20:	IF FSD.MODE = BYTE#0 THEN
		total_bytes := FSD.FILE_SIZE;
		X.NEW_FILE_SIZE := total_bytes + INT_TO_UDINT(idx);
		IF log_stop OR aw_aktiv THEN
			aw_aktiv := FALSE;
			FSD.MODE := BYTE#5; (* Datei schliessen *)
			(* ---------------- Debug-Message -----------------------*)
			(*IF _debug_enable THEN
				LOG_CL.NEW_MSG := 'FILE_XML2 - Close: [~2]';
				LOG_CL.PRINTF[2] := DT_TO_STRING(DTI);
				LOG_MSG();
			END_IF;*)
			(* -----------------------------------------------------------------*)
		END_IF;
		step_2 := 30;
	END_IF;

30:	IF FSD.MODE = BYTE#0 THEN (* Datei schliessen beendet *)
		IF log_stop THEN
			X.NEW_FILE_RTRIG := TRUE;
			log_stop := FALSE;
			SAVE_DATA.FN_REM := ''; (* remanenten Dateinamen löschen *)
		END_IF;
		step_2 := 00;
	END_IF;

END_CASE;

FS(FSD:=FSD,PT:=PT); (* FILE_SERVER *)

(* Fehlerauswertung *)
IF FSD.ERROR <> BYTE#0 THEN
	ERROR_C := BYTE_TO_DWORD(FSD.ERROR);
	ERROR_T := BYTE#1;
ELSIF X.UCB.BUF_DATA_LOST > UDINT#0 THEN
	ERROR_C := DWORD#2; (* Fehler: Bufferüberlauf - Datenmenge reduzieren *)
	ERROR_T := BYTE#6; 	(* Type: Buffer *)
ELSIF X.UCB.BUF_USED_MAX > USINT#90 THEN
	ERROR_C := DWORD#1; (* Warnung: Buffer auslastung > 90% *)
	ERROR_T := BYTE#6;	(* Type: Buffer *)
ELSE
	ERROR_C := DWORD#0;
	ERROR_T := BYTE#0;
END_IF;

trig_m_last := TRIG_M;

(* revision history
ks	25. july. 2011	rev 1.0
	original version

ks	16. apr. 2012	rev 1.1
	neuer überarbeiteter Code für automatisches File-open/close

ks	8. mar. 2016	rev 1.2
	nur einmal nach satellitenbausteinen scannen

ks	21. mar. 2016	rev 1.3
	prüfung auf freien bufferplatz hinzugefügt
	fehlermeldungen hinzugefügt

*)
          
END_FUNCTION_BLOCK

FUNCTION_BLOCK DLOG_STORE_MYSQL
  VAR_IN_OUT
    SQL_INFO : MYSQL_INFO;
    X : DLOG_DATA;
  END_VAR
  VAR_INPUT
    ENABLE : BOOL;
    TRIG_M : BOOL;
    TRIG_T : TIME;
    DTI : DT;
    URL : STRING(OSCAT_BASIC.STRING_LENGTH);
    DB_NAME : STRING(64);
    TB_NAME : STRING(64);
    AUTO_DELETE : UDINT;
    TIMEOUT : TIME;
    DNS_IP4 : DWORD;
  END_VAR
  VAR_OUTPUT
    ERROR_C : DWORD;
    ERROR_T : BYTE;
  END_VAR
  VAR
    UCB : UNI_CIRCULAR_BUFFER;
    MYSQL_CONTROL : MYSQL_CONTROL;
    trig_auto : BOOL;
    trig_tmp : BOOL;
    trig_m_last : BOOL;
    dti_last : DT := DATE_AND_TIME#2070-2-6-6:28:15;
    enable_last : BOOL;
    step : INT;
    idx : INT;
    n : USINT;
    snd_text : STRING(OSCAT_BASIC.STRING_LENGTH);
    snd_size : INT;
    sql_command : BYTE;
    next_step : INT;
    i1 : INT;
    i2 : INT;
    y : MYSQL_COM;
    del_dt : UDINT;
    del_start : BOOL;
    run : BOOL;
  END_VAR

            X.DTI := DTI; (* Datum / Zeit eintragen *)
X.CLOCK_TRIG := DTI <> dti_last;
dti_last := DTI;
trig_auto := FALSE;
IF X.CLOCK_TRIG THEN (* Impuls in jeder Sekunde *)
	del_start := DT_TO_UDINT(DTI) - del_dt > AUTO_DELETE AND AUTO_DELETE > UDINT#0;
	IF TRIG_T >= T#1000ms THEN (* automatischer Trigger *)
		trig_auto := DT_TO_UDINT(DTI) MOD (TIME_TO_UDINT(TRIG_T) / UDINT#1000) = UDINT#0;
	END_IF;
END_IF;
X.ADD_COM := 00;

CASE step OF

00:	IF ENABLE AND enable_last = FALSE THEN
		y.SQL_URL := URL;
		y.TIMEOUT := TIMEOUT;
		y.DNS_IP4 := DNS_IP4;
		y.SQL_CON := TRUE;

		X.UCB.D_MODE := 99; (* Buffer reset - Alles löschen *)
		UCB(DATA:=X.UCB);

		IF X.ID_MAX = USINT#0 THEN (* nur einmal nach Satellitenbausteinen scannen *)
			X.ADD_COM := 01; (* ADD INFO *)
			X.STORE_TYPE := BYTE#5; (* MySQL-Modus *)
		END_IF;

		step := 05;
	END_IF;

05:	X.ADD_COM := 02; (* ADD HEADER *)
	step := 10;

10:	IF SQL_INFO.SQL_CONNECTED THEN
		sql_command := BYTE#3; (* CREATE DATABASE IF NOT EXISTS `db_name` *)
		snd_text :=  CONCAT('CREATE DATABASE IF NOT EXISTS `' ,DB_NAME);
		snd_text :=  CONCAT(snd_text, '`');
		next_step := 20;
	END_IF;

20:	sql_command := BYTE#2; (* 0x02 COM_INIT_DB mysql_select_db *)
	snd_text := DB_NAME;
	next_step := 30;

30:	(* CREATE TABLE IF NOT EXISTS tb_name (Timestamp TIMESTAMP NULL DEFAULT CURRENT_TIMESTAMP, n1,n2) *)
	sql_command := BYTE#0;
	idx := 5;
	n := USINT#0;
	WHILE sql_command = BYTE#0 DO
		IF n = USINT#0 THEN
			snd_text := CONCAT('CREATE TABLE IF NOT EXISTS `', TB_NAME);
			snd_text := CONCAT(snd_text,'` (`ID` BIGINT NOT NULL AUTO_INCREMENT PRIMARY KEY ,');
			snd_text := CONCAT(snd_text,' store_timestamp TIMESTAMP NULL DEFAULT CURRENT_TIMESTAMP');
		ELSIF n <= X.ID_MAX THEN
			X.UCB.D_MODE := 12; (* Element lesen und löschen *)
			UCB(DATA:=X.UCB);
			snd_text := CONCAT(', `',X.UCB.D_STRING);
			CASE WORD_TO_INT(SHR(X.UCB.D_HEAD,8)) OF
			02:	snd_text := CONCAT(snd_text, '` FLOAT'); (* REAL *)
			06:	snd_text := CONCAT(snd_text, '` BOOL'); (* BOOL *)
			08:	snd_text := CONCAT(snd_text, '` INT'); (* DINT *)
			13:	snd_text := CONCAT(snd_text, '` DATETIME'); (* DT *)
			ELSE
				snd_text := CONCAT(snd_text, '` VARCHAR(80)'); (* STRING(80) *)
			END_CASE;
		ELSE
			snd_text := ')';
			sql_command := BYTE#3;
			snd_size := idx + LEN(snd_text);
			next_step := 40;
		END_IF;
		OSCAT_BASIC._STRING_TO_BUFFER(str:=snd_text,pos:=idx,pt:=ADR(y.S_BUF.BUFFER),size:=SIZEOF(y.S_BUF.BUFFER)); (* String in puffer kopieren *)
		idx := idx + LEN(snd_text);
		n := n + USINT#1;

		(*####################  DEBUG-MESSAGE  ###################################*)
		(*IF _debug_enable THEN
			LOG_CL.NEW_MSG := 'dlog_mysql: create >~1<';
			LOG_CL.PRINTF[1] := snd_text;
			LOG_MSG();
		END_IF;*)
		(*########################################################################*)
	END_WHILE;

40:	IF del_start THEN
		del_start := FALSE;
		sql_command := BYTE#3; (* DELETE FROM `tb_name` WHERE TIMESTAMPDIFF(SECOND, Timestamp, NOW()) > xxx *)
		snd_text := CONCAT('DELETE FROM `', TB_NAME);
		snd_text := CONCAT(snd_text, '` WHERE TIMESTAMPDIFF(SECOND, store_timestamp, NOW()) > ');
		snd_text := CONCAT(snd_text, UDINT_TO_STRING(AUTO_DELETE));
		next_step := 40;
		del_dt := DT_TO_UDINT(DTI);
		(*####################  DEBUG-MESSAGE  ###################################*)
		(*IF _debug_enable THEN
			LOG_CL.NEW_MSG := 'dlog_mysql: # delete time:~1 >~2<';
			LOG_CL.PRINTF[1] := UDINT_TO_STRING(AUTO_DELETE);
			LOG_CL.PRINTF[2] := snd_text;
			LOG_MSG();
		END_IF;*)
		(*########################################################################*)

         (* INSERT INTO `tb_name` VALUES (CURRENT_TIMESTAMP,  "n1","n2") *)
	ELSIF X.UCB.BUF_COUNT >= USINT_TO_INT(X.ID_MAX) AND step > 0 THEN (* Neue Datenreihe(n) vorhanden *)
		idx := 5;
		n := USINT#0;
		sql_command := BYTE#0;
		WHILE sql_command = BYTE#0 DO
			IF n = USINT#0 THEN
				snd_text := CONCAT('INSERT INTO `', TB_NAME);
				snd_text := CONCAT(snd_text,'` VALUES (NULL, CURRENT_TIMESTAMP');
			ELSIF n <= X.ID_MAX THEN
				X.UCB.D_MODE := 12; (* Element lesen und löschen *)
				UCB(DATA:=X.UCB);
				snd_text := CONCAT(', "',X.UCB.D_STRING);
				snd_text := CONCAT(snd_text, '"');
			ELSE
				snd_text := ')';
				sql_command := BYTE#3;
				snd_size := idx + LEN(snd_text);
				next_step := 40;
			END_IF;
			OSCAT_BASIC._STRING_TO_BUFFER(str:=snd_text,pos:=idx,pt:=ADR(y.S_BUF.BUFFER),size:=SIZEOF(y.S_BUF.BUFFER)); (* String in puffer kopieren *)
			idx := idx + LEN(snd_text);
			n := n + USINT#1;

			(*####################  DEBUG-MESSAGE  ###################################*)
			(*IF _debug_enable THEN
				LOG_CL.NEW_MSG := 'dlog_mysql: insert >~1<';
				LOG_CL.PRINTF[1] := snd_text;
				LOG_MSG();
			END_IF;*)
			(*########################################################################*)
		END_WHILE;
	END_IF;

	IF ENABLE THEN 	(* LOG-Trigger verarbeiten *)
		trig_tmp := (TRIG_M AND NOT trig_m_last) OR trig_auto OR X.ADD_DATA_REQ;

		IF trig_tmp THEN (* manueller, automatischer oder externer Trigger *)
			X.ADD_COM := 03; (* ADD DATA *)
			(* ---------------- Debug-Message -----------------------*)
			(*IF _debug_enable THEN
				LOG_CL.NEW_MSG := 'dlog_mysql: Trigger: DATE [~2]';
				LOG_CL.PRINTF[2] := DT_TO_STRING(DTI);
				LOG_MSG();
			END_IF;*)
			(* -----------------------------------------------------------------*)
		ELSE
			X.ADD_COM := 04;	(* ADD DATA REQ *)
		END_IF;
	ELSE
		y.SQL_CON := FALSE; (* MySQL Verbindung beenden *)
		step := 0;
	END_IF;
	X.ADD_DATA_REQ := FALSE;

(* ~~~~~~~~~~~~~~~~~~~~~~ *)

199:IF y.SQL_RCV_STATE = BYTE#1 THEN (* OK *)
		step := next_step;
	ELSIF y.SQL_RCV_STATE = BYTE#2 THEN  (* FEHLER *)
		step := 0;
	END_IF;

END_CASE;

(* ########################## *)
(* SQL-Kommando ausführen *)
IF sql_command > BYTE#0 THEN

	IF snd_size > 0 THEN
		y.S_BUF.SIZE := INT_TO_UINT(snd_size);
		snd_size := 0;
	ELSE
		OSCAT_BASIC._STRING_TO_BUFFER(str:=snd_text,pos:=5,pt:=ADR(y.S_BUF.BUFFER),size:=SIZEOF(y.S_BUF.BUFFER)); (* String in puffer kopieren *)
		y.S_BUF.SIZE := INT_TO_UINT(5 + LEN(snd_text));
		snd_text := '';
	END_IF;

	IF y.S_BUF.SIZE > SIZEOF(y.S_BUF.BUFFER) THEN (* buffer überlauf erkannt -> Abbruch *)
		y.S_BUF.SIZE := 0;
		sql_command := BYTE#0;
		y.SQL_CON := FALSE; (* MySQL Verbindung beenden *)
		step := 999; (* Dummy-Schritt *)
	ELSE

		i2 := UINT_TO_INT(y.S_BUF.SIZE) - 1; (* alle " zeichen mit ' ersetzen *)
		FOR i1 := 5 TO i2 DO
			IF y.S_BUF.BUFFER[i1] = BYTE#34 THEN
				y.S_BUF.BUFFER[i1] := BYTE#39;
			END_IF;
		END_FOR;
	
		y.S_BUF.BUFFER[4] := sql_command;
		y.SQL_PACKET_NO := BYTE#255;
		sql_command := BYTE#0;
		step := 199;
	END_IF;
END_IF;

(* ########################## *)

MYSQL_CONTROL(COM:= y, INFO:=SQL_INFO);

(* Fehlerauswertung *)
IF step = 999 THEN	(* Buffer überlauf *)
	ERROR_C := DWORD#3; (* Netzwerkbuffer überlauf *)
	ERROR_T := BYTE#6; 	(* Type: Buffer *)
ELSIF y.ERROR_T > BYTE#0 THEN	(* SQL Error *)
	ERROR_C := y.ERROR_C;
	ERROR_T := y.ERROR_T;
	step := 0;
ELSIF X.UCB.BUF_DATA_LOST > UDINT#0 THEN
	ERROR_C := DWORD#2; (* Fehler: Bufferüberlauf - Datenmenge reduzieren *)
	ERROR_T := BYTE#6; 	(* Type: Buffer *)
ELSIF X.UCB.BUF_USED_MAX > USINT#90 THEN
	ERROR_C := DWORD#1; (* Warnung: Buffer auslastung > 90% *)
	ERROR_T := BYTE#6;	(* Type: Buffer *)
ELSE
	ERROR_C := DWORD#0;
	ERROR_T := BYTE#0;
END_IF;



(* ########################## *)

trig_m_last := TRIG_M;
enable_last := ENABLE;
run := step > 0;

(* revision history
ks	20. apr. 2012	rev 1.0
	original version

ks	17. jan. 2014	rev 1.1
	DELTA Error 

ks	8. mar. 2016	rev 1.2
	nur einmal nach satellitenbausteinen scannen

ks	21. mar. 2016	rev 1.3
	prüfung auf bufferüberlauf und fehlermeldungen hinzugefügt

*)
          
END_FUNCTION_BLOCK

FUNCTION_BLOCK DLOG_STORE_RRD
  VAR_IN_OUT
    X : DLOG_DATA;
  END_VAR
  VAR_INPUT
    ENABLE : BOOL;
    TRIG_M : BOOL;
    TRIG_T : TIME;
    URL : STRING(OSCAT_BASIC.STRING_LENGTH);
    DTI : DT;
    SEP : BYTE;
    DNS_IP4 : DWORD;
    TIMEOUT : TIME;
  END_VAR
  VAR_OUTPUT
    ERROR_C : DWORD;
    ERROR_T : BYTE;
  END_VAR
  VAR
    UCB : UNI_CIRCULAR_BUFFER;
    IP_C : IP_C;  (* IP_Control Verwaltungsstruktur *)
    S_BUF : NETWORK_BUFFER;
    R_BUF : NETWORK_BUFFER;
    URL_DATA : url;
    DNS_CLIENT : DNS_CLIENT;
    HTTP_GET : HTTP_GET;
    IPC : IP_CONTROL;
    trig_auto : BOOL;
    trig_stored : BOOL;
    trig_tmp : BOOL;
    trig_m_last : BOOL;
    dti_last : DT := DATE_AND_TIME#2070-2-6-6:28:15;
    step_1 : INT;
    step_2 : INT;
    sep_char : STRING(1);
    url_query : STRING(OSCAT_BASIC.STRING_LENGTH);
    n : INT;
  END_VAR

            X.DTI := DTI; (* Datum / Zeit eintragen *)
X.CLOCK_TRIG := DTI <> dti_last;
dti_last := DTI;
trig_auto := FALSE;
IF X.CLOCK_TRIG THEN (* Impuls in jeder Sekunde *)
	IF TRIG_T >= T#1000ms THEN (* automatischer Trigger *)
		trig_auto := DT_TO_UDINT(DTI) MOD (TIME_TO_UDINT(TRIG_T) / UDINT#1000) = UDINT#0;
	END_IF;
END_IF;

CASE step_1 OF

00:	IF ENABLE THEN
		IF X.ID_MAX = USINT#0 THEN (* nur einmal nach Satellitenbausteinen scannen *)
			X.ADD_COM := 01; (* ADD INFO *)
			X.STORE_TYPE := BYTE#1; (* RRD-Modus *)
		END_IF;

		ERROR_T := BYTE#0;
		ERROR_C := DWORD#0;

		X.UCB.D_MODE := 99;
		UCB(DATA:=X.UCB); (* Buffer löschen *)

		URL_DATA:=STRING_TO_URL(STR:=URL,DEFAULT_PROTOCOL:='',DEFAULT_PATH:=''); (* URL zerlegen *)
		sep_char := OSCAT_BASIC.CHR_TO_STRING(SEP);
		url_query := URL_DATA.QUERY;
		step_1 := 30;

		(* ---------------- Debug-Message -----------------------*)
		(*IF _debug_enable THEN
			LOG_CL.NEW_MSG := 'FILE_RRD1 - Start: DATE [~2]';
			LOG_CL.PRINTF[2] := DT_TO_STRING(DTI);
			LOG_MSG();
		END_IF;*)
		(* -----------------------------------------------------------------*)

	END_IF;

30:	(* LOG-Trigger verarbeiten *)
	trig_tmp := (TRIG_M AND NOT trig_m_last) OR trig_auto OR X.ADD_DATA_REQ;

	IF ENABLE = FALSE THEN (* ENABLE = 0 -> Log Stop *)
		X.ADD_COM := 00;
		step_1 := 00;

		(* ---------------- Debug-Message -----------------------*)
		(*IF _debug_enable THEN
			LOG_CL.NEW_MSG := 'FILE_RRD1 - Stop: DATE [~2]';
			LOG_CL.PRINTF[2] := DT_TO_STRING(DTI);
			LOG_MSG();
		END_IF;*)
		(* -----------------------------------------------------------------*)

	ELSIF ENABLE THEN
		IF trig_tmp OR trig_stored THEN (* manueller, automatischer oder externer Trigger *)
			trig_stored := FALSE;
			X.ADD_COM := 03; (* ADD DATA *)
			(* ---------------- Debug-Message -----------------------*)
			(*IF _debug_enable THEN
				LOG_CL.NEW_MSG := 'FILE_RRD1 - Trig: DATE [~2]';
				LOG_CL.PRINTF[2] := DT_TO_STRING(DTI);
				LOG_MSG();
			END_IF;*)
			(* -----------------------------------------------------------------*)
		ELSE
			X.ADD_COM := 04;	(* ADD DATA REQ *)
		END_IF;
	END_IF;

END_CASE;
X.ADD_DATA_REQ := FALSE; (* externe Anforderung rücksetzen *)

(* ##################################### *)

CASE step_2 OF

00:	IF X.UCB.BUF_DATA_LOST > UDINT#0 THEN
		ERROR_C := DWORD#2; (* Fehler: Bufferüberlauf - Datenmenge reduzieren *)
		ERROR_T := BYTE#6; 	(* Type: Buffer *)
		step_2 := 100;
	ELSIF X.UCB.BUF_USED_MAX > USINT#90 THEN
		ERROR_C := DWORD#1; (* Warnung: Buffer auslastung > 90% *)
		ERROR_T := BYTE#6;	(* Type: Buffer *)
	END_IF;

	IF X.UCB.BUF_COUNT >= USINT_TO_INT(X.ID_MAX) THEN (* genug Einträge vorhanden *)
		URL_DATA.QUERY := url_query; (* original Query wiederherstellen *)
		n := 1;
		WHILE n <= USINT_TO_INT(X.ID_MAX) DO
			X.UCB.D_MODE := 12; (* Element lesen und löschen *)
			UCB(DATA:=X.UCB);
			IF n < USINT_TO_INT(X.ID_MAX) THEN (* Trennzeichen hinzufügen *)
				X.UCB.D_STRING := CONCAT(X.UCB.D_STRING,sep_char);
			END_IF;
			IF LEN(X.UCB.D_STRING) + LEN(URL_DATA.QUERY) <= OSCAT_BASIC.STRING_LENGTH THEN
				URL_DATA.QUERY := CONCAT(URL_DATA.QUERY,X.UCB.D_STRING); (* Query mit LOG-Daten ergänzen *)
				step_2 := 40;
			ELSE
				ERROR_T := BYTE#4; (* LOG-Daten können nicht in URL gepackt werden *)
				ERROR_C := DWORD#1;
				step_2 := 100;
			END_IF;
			n := n + 1;
		END_WHILE;;
	END_IF;

40:	IF DNS_CLIENT.DONE THEN
		step_2 := 60;
	ELSIF (DNS_CLIENT.ERROR > DWORD#0) THEN
		ERROR_C := DNS_CLIENT.ERROR; (* Fehlerbehandlung *)
		ERROR_T := BYTE#1;
		step_2 := 100;
	END_IF;

60:	IF HTTP_GET.DONE THEN
		n := UINT_TO_INT(HTTP_GET.BODY_START);
		IF R_BUF.BUFFER[n] <> BYTE#48 THEN (* ASCII '0' *)
			ERROR_C := DWORD#1;
			ERROR_T := BYTE#3;
		END_IF;
		step_2 := 100;

	ELSIF HTTP_GET.ERROR > DWORD#0 THEN (* Fehlerbehandlung *)
		ERROR_C := HTTP_GET.ERROR;
		ERROR_T := BYTE#2;
		step_2 := 100;
	END_IF;

100:	IF (NOT HTTP_GET.DONE) THEN (* UNLOCK HTTP DATA *)
		step_2 := SEL(ERROR_T = BYTE#0, 120,0);
	END_IF;

120:	IF NOT ENABLE THEN
		step_2 := 0;
	END_IF;

END_CASE;

HTTP_GET(IP_C:=IP_C,S_BUF:=S_BUF,R_BUF:=R_BUF,IP4:=DNS_CLIENT.IP4,GET:=step_2=60,MODE:=2,UNLOCK_BUF:=step_2=100,URL_DATA:=URL_DATA); (* HTTP_GET *)
DNS_CLIENT(IP_C:=IP_C, S_BUF:=S_BUF, R_BUF:=R_BUF, DOMAIN:=URL_DATA.DOMAIN, IP4_DNS:= DNS_IP4, ACTIVATE:=step_2=40); (* DNS-Client *)
IPC(IP:= 0, PORT:= 0 , TIME_OUT:= TIMEOUT, IP_C:= IP_C, S_BUF:= S_BUF, R_BUF:= R_BUF); (* IP_CONTROL *)

trig_m_last := TRIG_M;

(* revision history
ks	01. jan. 2011	rev 1.0
	original version

ks	13. may. 2011	rev 1.1
	ADD_DATA_REQ hinzugefügt

ks	26. july. 2011	rev 1.2
	code optimierung D_MODE 12 und bessere fehlerauswertung

ks	16. apr. 2012	rev 1.3
	neuer überarbeiteter Code

ks	21. mar. 2016	rev 1.4
	nur einmal nach satellitenbausteinen scannen und fehlermeldungen hinzugefügt

*)
          
END_FUNCTION_BLOCK

FUNCTION_BLOCK DLOG_STRING
  VAR_IN_OUT
    X : DLOG_DATA;
  END_VAR
  VAR_INPUT
    STR : STRING;
    COLUMN : STRING(40);
  END_VAR
  VAR
    UCB : UNI_CIRCULAR_BUFFER;
    id : WORD;
    str_last : STRING;
  END_VAR

            CASE x.ADD_COM OF

01:	(* ADD INFO *)
	X.ID_MAX := X.ID_MAX + USINT#1;
	id := WORD#16#0101; (* Quelltype STRING , Zieltype STRING *)
02:	(* ADD HEADER *)
	X.UCB.D_STRING := COLUMN;
	X.UCB.D_HEAD := id;
	X.UCB.D_MODE := 1;
	UCB(DATA:=X.UCB); (* Daten eintragen *)
03:	(* ADD DATA *)
	X.UCB.D_STRING := str_last;
	X.UCB.D_HEAD := id;
	X.UCB.D_MODE := 1;
	UCB(DATA:=X.UCB); (* Daten eintragen *)
END_CASE;
str_last := STR;

(* revision history
ks	01. jan. 2011	rev 1.0
	original version

ks	17. may. 2011	rev 1.1
	COLUMN STRING(40)

ks	25. july.   2011	rev 1.2
	neue head information

ks	19. apr.   2012	rev 1.3
	code neu überarbeitet
*)
          
END_FUNCTION_BLOCK

FUNCTION_BLOCK MYSQL_AUTH
  VAR_IN_OUT
    RUN : BOOL;
    PASSWORD : STRING(64);
    MESSAGE : ARRAY[0..19] OF BYTE;
    SCRAMBLE : ARRAY[0..19] OF BYTE;
  END_VAR
  VAR
    SHA1_STREAM : SHA1_STREAM;
    buf : ARRAY[0..63] OF BYTE;
    sha_mode : INT;
    step : INT;
    size : UDINT;
    pos : UDINT;
    i : INT;
    i2 : INT;
    scramble1 : ARRAY[0..19] OF BYTE;
    scramble2 : ARRAY[0..19] OF BYTE;
  END_VAR

            IF NOT RUN THEN RETURN; END_IF;
CASE step OF

0:	CASE sha_mode OF
	0:	sha_mode := 1; (* Initialisierung *)
		size := INT_TO_UDINT(LEN(PASSWORD));
		i2 := UDINT_TO_INT(size) - 1;
		FOR i := 0 TO 63 DO
			IF i <= i2 THEN
				buf[i] := OSCAT_BASIC.CODE(STR:=PASSWORD,POS:=i+1);
			ELSE
				buf[i] := BYTE#0;
			END_IF;
		END_FOR;

	3:	scramble1 := SCRAMBLE;
		sha_mode := 1; (* Initialisierung *)
		size := UDINT#20;
		FOR i := 0 TO 19 DO
			buf[i] := scramble1[i];
		END_FOR;
		step := 10;
	END_CASE;

10:	IF sha_mode = 3 THEN
		sha_mode := 1; (* Initialisierung *)
		scramble2 := SCRAMBLE;
		size := UDINT#40;
		FOR i := 0 TO 19 DO
			buf[i] := message[i];
			buf[i+20] := scramble2[i];
		END_FOR;
		step :=20;
	END_IF;

20:	IF sha_mode = 3 THEN
		sha_mode := 0; (* Stop *)
		FOR i:= 0 TO 19 DO
			SCRAMBLE[i] := SCRAMBLE[i] XOR scramble1[i];
		END_FOR;
		step :=0;
		RUN := FALSE;
	END_IF;
END_CASE;

SHA1_STREAM(SIZE:=size, MODE:=sha_mode, BUF:=buf, SHA1:=SCRAMBLE, POS=>pos);

(* revision history
ks	20. apr. 2012	rev 1.0
	original version

*)
          
END_FUNCTION_BLOCK

FUNCTION_BLOCK MYSQL_CONTROL
  VAR_IN_OUT
    COM : MYSQL_COM;
    INFO : MYSQL_INFO;
  END_VAR
  VAR
    IP_C : IP_C;
    URL_DATA : url;
    DNS_CLIENT : DNS_CLIENT;
    IPC : IP_CONTROL;
    step : INT;
    snd_step : INT;
    TON_WAIT : TON;
    last_step : INT;
    idx1 : INT;
    idx2 : INT;
    idx3 : INT;
    dw_tmp : DWORD;
    timeout1 : TIME;
    timeout2 : TIME;
    ip_c_red_disable : BOOL;
    auth_password : STRING(64);
    auth_run : BOOL;
    MYSQL_AUTH : MYSQL_AUTH;
    scramble1_buffer : ARRAY[0..19] OF BYTE;
    scramble2_buffer : ARRAY[0..19] OF BYTE;
    charset_number : BYTE := 16#8;
    max_packet_size : DWORD := 1024;
    client_flags : DWORD := 16#38601;
  END_VAR

            CASE step OF

00:	IF COM.SQL_CON THEN
		timeout1 := MAX(T#10s,COM.TIMEOUT);
		timeout2 := timeout1 + T#1s;
		INFO.SQL_ERROR := '';
		COM.ERROR_C := DWORD#0;
		COM.ERROR_T := BYTE#0;
		URL_DATA := STRING_TO_URL(STR:=COM.SQL_URL,DEFAULT_PROTOCOL:='',DEFAULT_PATH:='/');
		step := 10;
	END_IF;

10:	IF DNS_CLIENT.DONE THEN
		step := 20;
	ELSIF DNS_CLIENT.ERROR <> DWORD#0 THEN
		COM.ERROR_C := DNS_CLIENT.ERROR;
		COM.ERROR_T := BYTE#1;
		step := 980;
	END_IF;

20:	(* MySQL Steuerkanal einrichten *)
	IF URL_DATA.PORT = WORD#0 THEN
		URL_DATA.PORT := WORD#3306; (* Standard Port *)
	END_IF;
	IP_C.C_PORT := URL_DATA.PORT; (* Portnummer eintragen *)
  	IP_C.C_IP := DNS_CLIENT.IP4; (* IP eintragen *)
  	IP_C.C_MODE := BYTE#0; (* Mode: TCP+ACTIV+PORT *)
  	IP_C.TIME_RESET := TRUE; (* Zeitueberwachung rücksetzen *)
  	IP_C.C_ENABLE := TRUE; (* Verbindungsaufbau freigeben *)
  	IP_C.R_OBSERVE := TRUE; (* Empfangsueberwachung *)
	COM.R_BUF.SIZE := UINT#0;
	COM.SQL_RCV_STATE := BYTE#0;
	step := 30;

30:	IF COM.SQL_RCV_STATE = BYTE#1 THEN
		INFO.SERVER_PROTOCOL_VERSION := COM.R_BUF.BUFFER[4];

		(* ende markierung von string server_version suchen *)
		idx2 := UINT_TO_INT(COM.R_BUF.SIZE) - 1;
		FOR idx1 := 5 TO idx2 DO
			IF COM.R_BUF.BUFFER[idx1] = BYTE#0 THEN EXIT; END_IF;
		END_FOR;
		idx1 := idx1 + 5; (* terminierung und thread-id überspringen *)

		FOR idx2:=0 TO 7 DO	(* Byte 0-7 *)
			scramble1_buffer[idx2] := COM.R_BUF.BUFFER[idx1];
			idx1 := idx1 + 1;
		END_FOR;
		idx1 := idx1 + 1;
		idx2 := idx1 + 1;
		INFO.SERVER_CAPABILITIES := OSCAT_BASIC.WORD_OF_BYTE(COM.R_BUF.BUFFER[idx2], COM.R_BUF.BUFFER[idx1]);
		idx1 := idx1 + 2;
		INFO.SERVER_LANGUAGE := COM.R_BUF.BUFFER[idx1];
		idx1 := idx1 + 1;
		idx2 := idx1 + 1;
		INFO.SERVER_STATUS := OSCAT_BASIC.WORD_OF_BYTE(COM.R_BUF.BUFFER[idx2], COM.R_BUF.BUFFER[idx1]);
		idx1 := idx1 + 15;

		FOR idx2:=8 TO 19 DO	(* Byte 8-19 *)
			scramble1_buffer[idx2] := COM.R_BUF.BUFFER[idx1];
			idx1 := idx1 + 1;
		END_FOR;

		IF INFO.SERVER_PROTOCOL_VERSION < BYTE#10 THEN  (* Error: protocol version zu niedrig *)
			COM.ERROR_T := BYTE#2;
			COM.ERROR_C := DWORD#1;
			step := 980;
		ELSIF URL_DATA.PASSWORD = '' THEN
			step := 50;
		ELSE
			auth_password := URL_DATA.PASSWORD;
			auth_run := TRUE;
			step := 40;
		END_IF;
	END_IF;

40:	MYSQL_AUTH(RUN:= auth_run,PASSWORD:= auth_password ,MESSAGE:= scramble1_buffer,SCRAMBLE:= scramble2_buffer);
	IF NOT auth_run THEN
		step := 50;
	END_IF;

50: (* Client Authentication Packet *)
	(* Byte 0-3 werden später eingetragen *)
	COM.S_BUF.BUFFER[04] := OSCAT_BASIC.BYTE_OF_DWORD(client_flags, BYTE#0); (* client_flags *)
	COM.S_BUF.BUFFER[05] := OSCAT_BASIC.BYTE_OF_DWORD(client_flags, BYTE#1);
	COM.S_BUF.BUFFER[06] := OSCAT_BASIC.BYTE_OF_DWORD(client_flags, BYTE#2);
	COM.S_BUF.BUFFER[07] := OSCAT_BASIC.BYTE_OF_DWORD(client_flags, BYTE#3);
	COM.S_BUF.BUFFER[08] := OSCAT_BASIC.BYTE_OF_DWORD(max_packet_size, BYTE#0); (* max_packet_size *)
	COM.S_BUF.BUFFER[09] := OSCAT_BASIC.BYTE_OF_DWORD(max_packet_size, BYTE#1);
	COM.S_BUF.BUFFER[10] := OSCAT_BASIC.BYTE_OF_DWORD(max_packet_size, BYTE#2);
	COM.S_BUF.BUFFER[11] := OSCAT_BASIC.BYTE_OF_DWORD(max_packet_size, BYTE#3);
	COM.S_BUF.BUFFER[12] := charset_number; (* charset_number *)
	FOR idx1 := 13 TO 35 DO (* 23 bytes filler always 0x00.. *)
		COM.S_BUF.BUFFER[idx1] := BYTE#0;
	END_FOR;
	idx3 := LEN(URL_DATA.USER);
	FOR idx2 :=1 TO idx3 DO
		COM.S_BUF.BUFFER[idx1] := OSCAT_BASIC.CODE(URL_DATA.USER, idx2);
		idx1 := idx1 + 1;
	END_FOR;
	COM.S_BUF.BUFFER[idx1] := BYTE#0; (* String terminierung eintragen *)
	idx1 := idx1 + 1;
	IF LEN(URL_DATA.PASSWORD) = 0 THEN
		COM.S_BUF.BUFFER[idx1] := BYTE#0; (* scramble_buff length *)
	ELSE
		COM.S_BUF.BUFFER[idx1] := BYTE#20; (* scramble_buff length *)
		FOR idx2 :=0 TO 19 DO
			idx1 := idx1 + 1;
			COM.S_BUF.BUFFER[idx1] := scramble2_buffer[idx2];
		END_FOR;
	END_IF;
	COM.S_BUF.SIZE  := INT_TO_UINT(idx1 + 1); (* Sendelänge eintragen *)

	step := 60;

60:	IF COM.SQL_RCV_STATE = BYTE#1 THEN
		INFO.SQL_CONNECTED := TRUE;
		step := 300;
	END_IF;

(* ================================================== *)

300:	step := SEL(COM.SQL_CON,700,310); (* Schritt-Selektion *)

310:	step := 300; (* dummy step *)

(* ================================================== *)

700: (* COM_QUIT *)
	COM.S_BUF.BUFFER[04] := BYTE#1; (* 0x01 COM_QUIT mysql_close *)
	COM.S_BUF.SIZE := UINT#5; (* Sendelänge eintragen *)
	COM.SQL_PACKET_NO := BYTE#255;
	ip_c_red_disable := TRUE;
	step := 710;

710:	IF IP_C.C_STATE = BYTE#0 THEN (* Verbindung durch SQL-Server beendet ? *)
		step := 980;
	END_IF;

(* ================================================== *)

980:IP_C.C_ENABLE := FALSE; (* MYSQL Steuerkanal schliessen *)
	ip_c_red_disable := FALSE;
	INFO.SQL_CONNECTED := FALSE;
	COM.SQL_CON := FALSE;
	COM.S_BUF.SIZE := UINT#0;
	COM.R_BUF.SIZE := UINT#0;
	snd_step := 0;
	step := 990;
	(*####################  DEBUG-MESSAGE  ###################################*)
	(*IF _debug_enable THEN
		LOG_CL.NEW_MSG := 'QUIT: ERROR CODE >~1< TYPE >~2<';
		LOG_CL.PRINTF[1] := DWORD_TO_STRH(COM.ERROR_C);
		LOG_CL.PRINTF[2] := BYTE_TO_STRING(COM.ERROR_T);
		LOG_MSG();
	END_IF;*)
	(*########################################################################*)

990:IF IP_C.C_STATE = BYTE#0 THEN
		step := 0;
	END_IF;

END_CASE;

(* ++++++++++++++++++++++++++++++++++++++++++++++++++++++++++ *)

IF step >= 30 THEN
	IF COM.R_BUF.SIZE >= UINT#3 AND COM.SQL_RCV_STATE = BYTE#0 THEN (* Daten wurden empfangen ? *)
		IF DWORD_TO_UINT(OSCAT_BASIC.DWORD_OF_BYTE(BYTE#0, COM.R_BUF.BUFFER[2], COM.R_BUF.BUFFER[1], COM.R_BUF.BUFFER[0])) + UINT#4 = COM.R_BUF.SIZE THEN
			COM.SQL_PACKET_NO := COM.R_BUF.BUFFER[3];
			IF COM.R_BUF.BUFFER[4] = BYTE#16#FF THEN
				idx2 := 13; (* Error String - Erstes Zeichen *)
				idx3 := UINT_TO_INT(COM.R_BUF.SIZE) - 1; (* Error String - Letztes Zeichen *)
				FOR idx1 := idx2 TO idx3 DO (* alle ' durch ´ ersetzen *)
					IF COM.R_BUF.BUFFER[idx1] = BYTE#39 THEN
						COM.R_BUF.BUFFER[idx1] := BYTE#96;
					END_IF;
				END_FOR;
				INFO.SQL_ERROR := OSCAT_BASIC.BUFFER_TO_STRING(PT:=ADR(COM.R_BUF.BUFFER),SIZE:=COM.R_BUF.SIZE,START:=INT_TO_UINT(idx2),STOP:=INT_TO_UINT(idx3));
				COM.ERROR_T := BYTE#3;
				COM.ERROR_C := OSCAT_BASIC.DWORD_OF_BYTE(BYTE#0,BYTE#0,COM.R_BUF.BUFFER[6], COM.R_BUF.BUFFER[5]);
				COM.SQL_RCV_STATE := BYTE#2;
				COM.R_BUF.SIZE := UINT#0; (* Empfangsbuffer nach Fehler rücksetzen *)
				step := 980;
			ELSE
				COM.SQL_RCV_STATE := BYTE#1;
				IP_C.R_OBSERVE := FALSE;

				(*####################  DEBUG-MESSAGE  ###################################*)
				(*IF _debug_enable THEN
					LOG_CL.NEW_MSG := 'RCV: size >~1<';
					LOG_CL.PRINTF[1] := UINT_TO_STRING(COM.R_BUF.SIZE);
					LOG_MSG();
				END_IF;*)
				(*########################################################################*)
			END_IF;
		END_IF;
	END_IF;
END_IF;

(* automatisches Datensenden *)

CASE snd_step OF

00:	IF step >= 20 AND COM.S_BUF.SIZE > UINT#0 THEN
		dw_tmp := UINT_TO_DWORD(COM.S_BUF.SIZE - UINT#4); (* packet_length *)
		COM.S_BUF.BUFFER[0] := OSCAT_BASIC.BYTE_OF_DWORD(dw_tmp, BYTE#0);
		COM.S_BUF.BUFFER[1] := OSCAT_BASIC.BYTE_OF_DWORD(dw_tmp, BYTE#1);
		COM.S_BUF.BUFFER[2] := 0;
		COM.SQL_PACKET_NO := COM.SQL_PACKET_NO + 1;
		COM.S_BUF.BUFFER[3] := COM.SQL_PACKET_NO;

		IP_C.R_OBSERVE := TRUE;
		COM.R_BUF.SIZE := UINT#0; (* Empfangsbuffer rücksetzen *)
		COM.SQL_RCV_STATE := BYTE#0;

	        (*####################  DEBUG-MESSAGE  ###################################*)
	        (*IF _debug_enable THEN
	          LOG_CL.NEW_MSG := 'SND: size >~1<';
	          LOG_CL.PRINTF[1] := UINT_TO_STRING(COM.S_BUF.SIZE);
	          LOG_MSG();
	        END_IF;*)
	        (*########################################################################*)

		snd_step := 10;
	END_IF;

10:	IF COM.S_BUF.SIZE = UINT#0 THEN (* warten bis alle daten gesendet sind *)
		snd_step := 0;
	END_IF;

END_CASE;

(* Globale Fehlerbehandlung für Haupt-Routine *)
IF COM.ERROR_T = BYTE#0 AND step > 20 THEN (* noch kein Fehler gespeichert und Hauptroutine aktiv *)
	IF IP_C.ERROR > DWORD#0 AND IP_C.C_ENABLE AND NOT IP_C.TIME_RESET THEN  (* IP Control *)
		IF ip_c_red_disable = FALSE OR IP_C.ERROR <> DWORD#16#FD000000 THEN
			COM.ERROR_C := IP_C.ERROR;
			COM.ERROR_T := BYTE#2;
			step := 980;
		END_IF;
	END_IF;
END_IF;

IF TON_WAIT.Q THEN (* Ablaufstörung - Schrittkette *)
	COM.ERROR_C := INT_TO_DWORD(step); (* aktuellen Schritt eintragen *)
	COM.ERROR_T := BYTE#5;
	step := 980;
END_IF;

(* ######################################################## *)

DNS_CLIENT(IP_C:=IP_C, S_BUF:=COM.S_BUF, R_BUF:=COM.R_BUF, DOMAIN:=URL_DATA.DOMAIN, IP4_DNS:= COM.DNS_IP4, ACTIVATE:=step=10); (* DNS-Client *)
IPC(IP:= DWORD#0, PORT:= WORD#0 , TIME_OUT:= timeout1, IP_C:= IP_C, S_BUF:= COM.S_BUF, R_BUF:= COM.R_BUF); (* MYSQL Steuerkanal *)

TON_WAIT(IN:=step = last_step AND step > 0,PT:=timeout2);
last_step := step;

(* revision history
ks	20. apr. 2012	rev 1.0
	original version
ks	14. oct. 2013	rev 1.1
	DNS_CLIENT Fehler durch zugriffskonflikt zwischen dns_client und mySQL auf S_BUF

*)
          
END_FUNCTION_BLOCK

PROGRAM BASE64_DEMO
  VAR
    text1 : STRING(144) := '<4036.1076324381@guildenstern.zeitform.de>';
    text2 : STRING(192);
    text3 : STRING(144);
    BASE64_DECODE_STR : BASE64_DECODE_STR;
    BASE64_ENCODE_STR : BASE64_ENCODE_STR;
    start : BOOL := TRUE;
    done1 : BOOL;
    done2 : BOOL;
  END_VAR

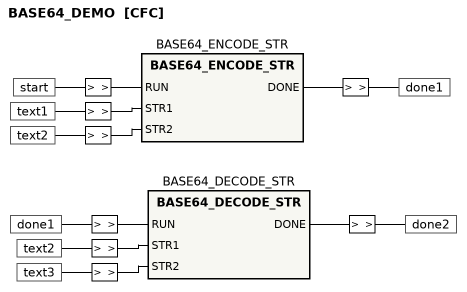
(* CFC diagram, written out as Structured Text *)
BASE64_ENCODE_STR(RUN := start, STR1 := text1, STR2 := text2);
done1 := BASE64_ENCODE_STR.DONE;
BASE64_DECODE_STR(RUN := done1, STR1 := text2, STR2 := text3);
done2 := BASE64_DECODE_STR.DONE;
END_PROGRAM

PROGRAM CSV_PARSER_BUF_DEMO
  VAR CONSTANT
    line_cnt : INT := 2;
    col_cnt : INT := 4;
  END_VAR
  VAR
    CPB : CSV_PARSER_BUF;
    FS : FILE_SERVER;
    FSD : FILE_SERVER_DATA;
    PT : NETWORK_BUFFER;
    sep : BYTE;
    value : STRING(OSCAT_BASIC.STRING_LENGTH);
    step : INT;
    result : BYTE;
    offset : UDINT;
    run : BYTE;
    done : BOOL;
    value_real : REAL;
    cnt : INT;
    line : INT;
    idx : INT;
    data : ARRAY[1..line_cnt, 1..col_cnt] OF REAL;
  END_VAR

            (* Demo-Programm: CSV-Datei mittels Enumeration auswerten
die groesse des arrays kann mittels konstanten line_cnt und col_cnt angepasst werden

 ----- den nachfolgenden Textblock als datei "csv.txt" auf der sps ablegen ---
10.45,20,30,40.8
115,3450.2123,456,123.1
---------------------------------------------------------------------------------*)

CASE step OF

00:	IF NOT done THEN
	 	(* File_Daten einrichten  *)
		FSD.FILENAME := 'csv.txt'; (* Dateiname *)
		FSD.MODE := 1; (* vorhandene Datei zum lesen öffnen *)
		FSD.OFFSET := 0; (* Start bei Dateianfang *)
		PT.SIZE := 65535; (* maximale länge einlesen *)
		step := 10;
	END_IF;

10:	IF FSD.MODE = 0 THEN (* Datei geöffnet ? *)
		OFFSET := 0; (* Start Offset vorgeben *)
		sep :=44; (* Trennzeichen , *)
		run := 1; (* Element suchen *)
		cnt := 0;
		step := 20;
	END_IF;

20:	IF run = 0 THEN
		(* ---------------------- Debug-Message ----------------------------*)
		(*IF _debug_enable THEN
			LOG_CL.NEW_MSG := 'CPFD: /value >~2< /offset ~3 /Run ~4 /Result ~5';
			LOG_CL.PRINTF[2] := value;
			LOG_CL.PRINTF[3] := UDINT_TO_STRING(OFFSET);
			LOG_CL.PRINTF[4] := BYTE_TO_STRING(run);
			LOG_CL.PRINTF[5] := BYTE_TO_STRING(result);
			LOG_MSG();
		END_IF;*)
		(* -----------------------------------------------------------------*)

		run := 1; (*  nächstes Element suchen  *)

		IF result = 1 OR result = 2 THEN
			(* automatische konvertierung in real ausführen *)
			IF LEN(value) <= 20 THEN
				value_real := OSCAT_BASIC.FLOAT_TO_REAL(FLT:=value);
			ELSE
				value_real := 0.0;
			END_IF;

			cnt := cnt + 1;
			IF cnt <= line_cnt * col_cnt THEN
				line := (cnt / col_cnt) + 1;
				idx := (cnt MOD col_cnt);
				data[line,idx] := value_real; (* Daten in Array eintragen *)
			END_IF;

		ELSIF result = 10 THEN (* nichts mehr gefunden *)
			run := 0; (* keine weitere INI Auswertung erwünscht *)
			FSD.MODE := 5; (* Datei schliessen *)
			step := 30;
		END_IF;
	END_IF;

30:	IF FSD.MODE = 0 THEN (* Datei geschlossen ? *)
		step := 0;
		done := TRUE;
	END_IF;

END_CASE;

CPB(SEP:=sep,RUN:=run,OFFSET:=OFFSET,VALUE:=value,PT:=PT,RESULT=>result); (* CSV PARAMETER BUF *)
FS(FSD:=FSD,PT:=PT); (* FILE_SERVER *)
          
END_PROGRAM

PROGRAM CSV_PARSER_FILE_DEMO
  VAR CONSTANT
    line_cnt : INT := 2;
    col_cnt : INT := 4;
  END_VAR
  VAR
    CPF : CSV_PARSER_FILE;
    FS : FILE_SERVER;
    FSD : FILE_SERVER_DATA;
    PT : NETWORK_BUFFER;
    filename : STRING;
    value : STRING(OSCAT_BASIC.STRING_LENGTH);
    sep : BYTE;
    step : INT;
    result : BYTE;
    offset : UDINT;
    run : BYTE;
    done : BOOL;
    value_real : REAL;
    cnt : INT;
    line : INT;
    idx : INT;
    data : ARRAY[1..line_cnt, 1..col_cnt] OF REAL;
  END_VAR

            (* Demo-Programm: CSV-Datei mittels Enumeration auswerten

die groesse des arrays kann mittels konstanten line_cnt und col_cnt angepasst werden

 ----- den nachfolgenden Textblock als datei "csv.txt" auf der sps ablegen ---
10.45,20,30,40.8
115,3450.2123,456,123.1
---------------------------------------------------------------------------------*)

CASE step OF

00:	IF NOT done THEN
		filename := 'csv.txt'; (* File_Daten einrichten *)
		OFFSET := 0; (* Start Offset vorgeben *)
		sep :=44; (* Trennzeichen , *)
		run := 1; (* Element suchen *)
		cnt := 0;
		step := 20;
	END_IF;

20:	IF run = 0 THEN (* kein Befehl mehr aktiv ? *)
		(* ---------------------- Debug-Message ----------------------------*)
		(*IF _debug_enable THEN
			LOG_CL.NEW_MSG := 'CPFD: /value >~2< /offset ~3 /Run ~4 /Result ~5';
			LOG_CL.PRINTF[2] := value;
			LOG_CL.PRINTF[3] := UDINT_TO_STRING(OFFSET);
			LOG_CL.PRINTF[4] := BYTE_TO_STRING(run);
			LOG_CL.PRINTF[5] := BYTE_TO_STRING(result);
			LOG_MSG();
		END_IF;*)
		(* -----------------------------------------------------------------*)

		run := 1; (*  nächstes Element suchen  *)

		IF result = 1 OR result = 2 THEN
			(* automatische konvertierung in real ausführen *)
			IF LEN(value) <= 20 THEN
				value_real := OSCAT_BASIC.FLOAT_TO_REAL(FLT:=value);
			ELSE
				value_real := 0.0;
			END_IF;

			cnt := cnt + 1;
			IF cnt <= line_cnt * col_cnt THEN
				line := (cnt / col_cnt) + 1;
				idx := (cnt MOD col_cnt);
				data[line,idx] := value_real; (* Daten in Array eintragen *)
			END_IF;

		ELSIF result = 10 THEN (* nichts mehr gefunden *)
			run := 0; (* keine weitere INI Auswertung erwünscht *)
			FSD.MODE := 5; (* Datei schliessen *)
			step := 30;
		END_IF;
	END_IF;

30:	IF FSD.MODE = 0 THEN (* Befehl Datei schliessen beendet *)
		step := 0;
		done := TRUE;
	END_IF;

END_CASE;

CPF(SEP:=sep,FILENAME:=FILENAME,FSD:=FSD,RUN:=run,OFFSET:=OFFSET,VALUE:=value,PT:=PT,RESULT=>result); (* CSV PARAMETER FILE *)
FS(FSD:=FSD,PT:=PT); (* FILE_SERVER *)
          
END_PROGRAM

PROGRAM DLOG_FILE_CSV_DEMO
  VAR
    cur_dt : DT;
    enable : BOOL := TRUE;
    trig_t : TIME := TIME#5s0ms;
    trig_m : BOOL;
    error_c : DWORD;
    error_t : BYTE;
    auto_close : TIME := TIME#10s0ms;
    x1 : DLOG_DT;
    x2 : DLOG_REAL;
    x3 : DLOG_DINT;
    x4 : DLOG_BOOL;
    x5 : DLOG_STRING;
    x : DLOG_DATA;
    RTC_2 : oscat_basic.RTC_2;
    DLOG_STORE_FILE_CSV : DLOG_STORE_FILE_CSV;
    GEN_SIN_1 : oscat_basic.GEN_SIN;
    COUNT_DR : oscat_basic.COUNT_DR;
  END_VAR
  VAR RETAIN
    save_data : DLOG_SAVE;
  END_VAR

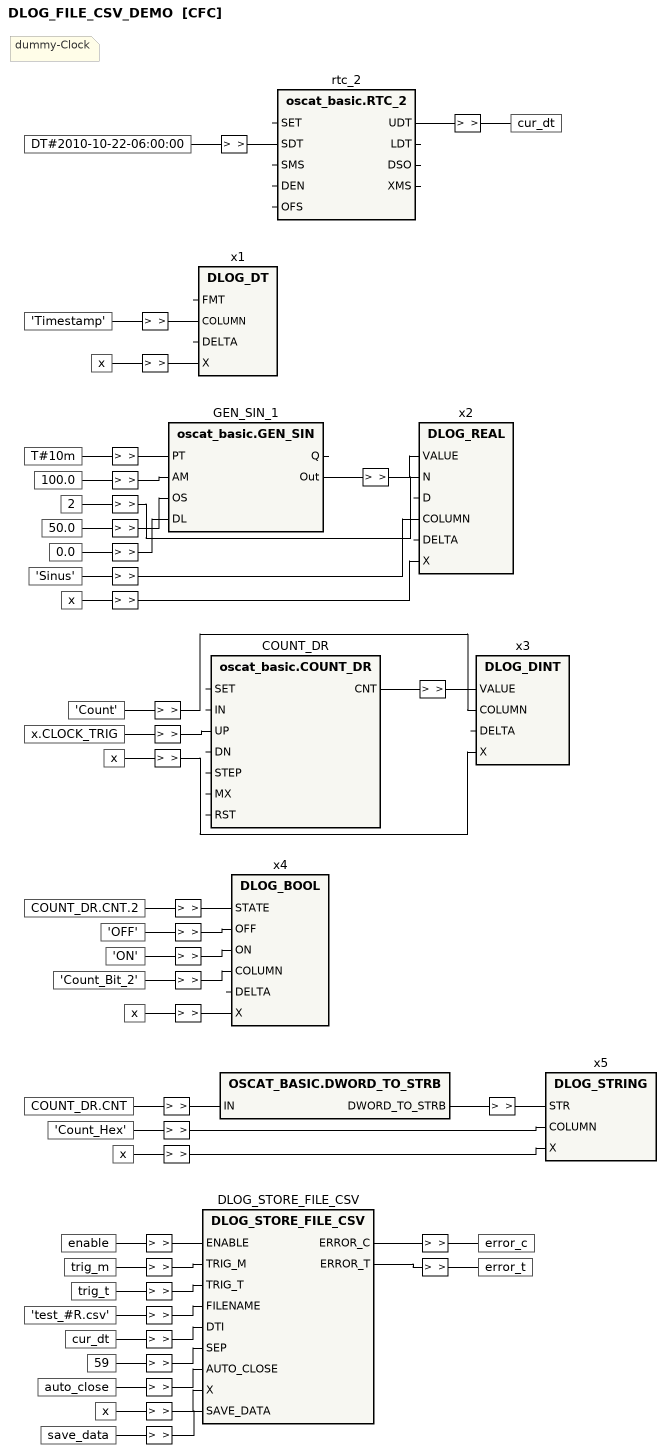
(* CFC diagram, written out as Structured Text *)
(* dummy-Clock *)
rtc_2(SDT := DT#2010-10-22-06:00:00);
cur_dt := rtc_2.UDT;
x1(COLUMN := 'Timestamp', X := x);
GEN_SIN_1(PT := T#10m, AM := 100.0, OS := 50.0, DL := 0.0);
x2(VALUE := GEN_SIN_1.Out, N := 2, COLUMN := 'Sinus', X := x);
COUNT_DR(UP := x.CLOCK_TRIG);
x3(VALUE := COUNT_DR.CNT, COLUMN := 'Count', X := x);
x4(STATE := COUNT_DR.CNT.2, OFF := 'OFF', ON := 'ON', COLUMN := 'Count_Bit_2', X := x);
x5(STR := OSCAT_BASIC.DWORD_TO_STRB(COUNT_DR.CNT), COLUMN := 'Count_Hex', X := x);
DLOG_STORE_FILE_CSV(ENABLE := enable, TRIG_M := trig_m, TRIG_T := trig_t, FILENAME := 'test_#R.csv', DTI := cur_dt, SEP := 59, AUTO_CLOSE := auto_close, X := x, SAVE_DATA := save_data);
error_c := DLOG_STORE_FILE_CSV.ERROR_C;
error_t := DLOG_STORE_FILE_CSV.ERROR_T;
END_PROGRAM

PROGRAM DLOG_FILE_CSV_FTP_DEMO
  VAR
    cur_dt : DT;
    enable : BOOL := TRUE;
    trig_t : TIME := TIME#5s0ms;
    trig_m : BOOL;
    error_c : DWORD;
    error_t : BYTE;
    auto_close : TIME := TIME#10s0ms;
    x1 : DLOG_DT;
    x2 : DLOG_REAL;
    x3 : DLOG_DINT;
    x4 : DLOG_BOOL;
    x5 : DLOG_STRING;
    x : DLOG_DATA;
    RTC_2 : oscat_basic.RTC_2;
    DLOG_STORE_FILE_CSV : DLOG_STORE_FILE_CSV;
    GEN_SIN_1 : oscat_basic.GEN_SIN;
    COUNT_DR : oscat_basic.COUNT_DR;
    DLOG_FILE_TO_FTP : DLOG_FILE_TO_FTP;
    ftp_done : BOOL;
    ftp_busy : BOOL;
    ftp_error_c : DWORD;
    ftp_error_t : BYTE;
    ftp_url : STRING := 'ftp://581920:123456@oscat.atwebpages.com:2000/subordner/';
    ftp_activ : BOOL := FALSE;
    ftp_delete : BOOL := TRUE;
    ftp_retry : INT := 0;
    ftp_retry_time : TIME := TIME#1m0s0ms;
    ftp_timeout : TIME := TIME#30s0ms;
  END_VAR
  VAR RETAIN
    save_data : DLOG_SAVE;
  END_VAR

(* CFC diagram, written out as Structured Text *)
(* dummy-Clock *)
rtc_2(SDT := DT#2010-10-22-06:00:00);
cur_dt := rtc_2.UDT;
x1(COLUMN := 'Timestamp', X := x);
GEN_SIN_1(PT := T#10m, AM := 100.0, OS := 50.0, DL := 0.0);
x2(VALUE := GEN_SIN_1.Out, N := 2, COLUMN := 'Sinus', X := x);
COUNT_DR(UP := x.CLOCK_TRIG);
x3(VALUE := COUNT_DR.CNT, COLUMN := 'Count', X := x);
x4(STATE := COUNT_DR.CNT.2, OFF := 'OFF', ON := 'ON', COLUMN := 'Count_Bit_2', X := x);
x5(STR := OSCAT_BASIC.DWORD_TO_STRB(COUNT_DR.CNT), COLUMN := 'Count_Hex', X := x);
DLOG_STORE_FILE_CSV(ENABLE := enable, TRIG_M := trig_m, TRIG_T := trig_t, FILENAME := 'test_#R.csv', DTI := cur_dt, SEP := 59, AUTO_CLOSE := auto_close, X := x, SAVE_DATA := save_data);
error_c := DLOG_STORE_FILE_CSV.ERROR_C;
error_t := DLOG_STORE_FILE_CSV.ERROR_T;
DLOG_FILE_TO_FTP(FTP_URL := ftp_url, FTP_ACTIV := ftp_activ, FILE_DELETE := ftp_delete, TIMEOUT := ftp_timeout, RETRY := ftp_retry, RETRY_TIME := ftp_retry_time, DNS_IP4 := oscat_basic.DWORD_OF_BYTE(8, 8, 8, 8), PLC_IP4 := oscat_basic.DWORD_OF_BYTE(192, 168, 178, 025), X := x);
ftp_done := DLOG_FILE_TO_FTP.DONE;
ftp_busy := DLOG_FILE_TO_FTP.BUSY;
ftp_error_c := DLOG_FILE_TO_FTP.ERROR_C;
ftp_error_t := DLOG_FILE_TO_FTP.ERROR_T;
END_PROGRAM

PROGRAM DLOG_FILE_CSV_SMTP_DEMO
  VAR
    cur_dt : DT;
    enable : BOOL := TRUE;
    trig_t : TIME := TIME#5s0ms;
    trig_m : BOOL;
    error_c : DWORD;
    error_t : BYTE;
    auto_close : TIME := TIME#10s0ms;
    x1 : DLOG_DT;
    x2 : DLOG_REAL;
    x3 : DLOG_DINT;
    x4 : DLOG_BOOL;
    x5 : DLOG_STRING;
    x : DLOG_DATA;
    RTC_2 : oscat_basic.RTC_2;
    DLOG_STORE_FILE_CSV : DLOG_STORE_FILE_CSV;
    GEN_SIN_1 : oscat_basic.GEN_SIN;
    COUNT_DR : oscat_basic.COUNT_DR;
    DLOG_FILE_TO_SMTP : DLOG_FILE_TO_SMTP;
    smtp_timeout : TIME := TIME#30s0ms;
    smtp_error_t : BYTE;
    smtp_error_c : DWORD;
    smtp_busy : BOOL;
    smtp_done : BOOL;
    smtp_dti : DT;
    smtp_dti_offset : INT := 60;
    smtp_server : STRING := '110876022:oscat123456@mail.gmx.net';
    smtp_mailfrom : STRING := 'oscat@gmx.net;Station_01';
    smtp_mailto : STRING(OSCAT_BASIC.STRING_LENGTH) := 'oscat@gmx.net';
    smtp_subject : STRING := 'Das ist der Betreff';
    smtp_body : STRING(OSCAT_BASIC.STRING_LENGTH) := 'Das ist der Email-Text';
    smtp_delete : BOOL := TRUE;
    smtp_retry : INT := 0;
    smtp_retry_time : TIME := TIME#1m0s0ms;
  END_VAR
  VAR RETAIN
    save_data : DLOG_SAVE;
  END_VAR

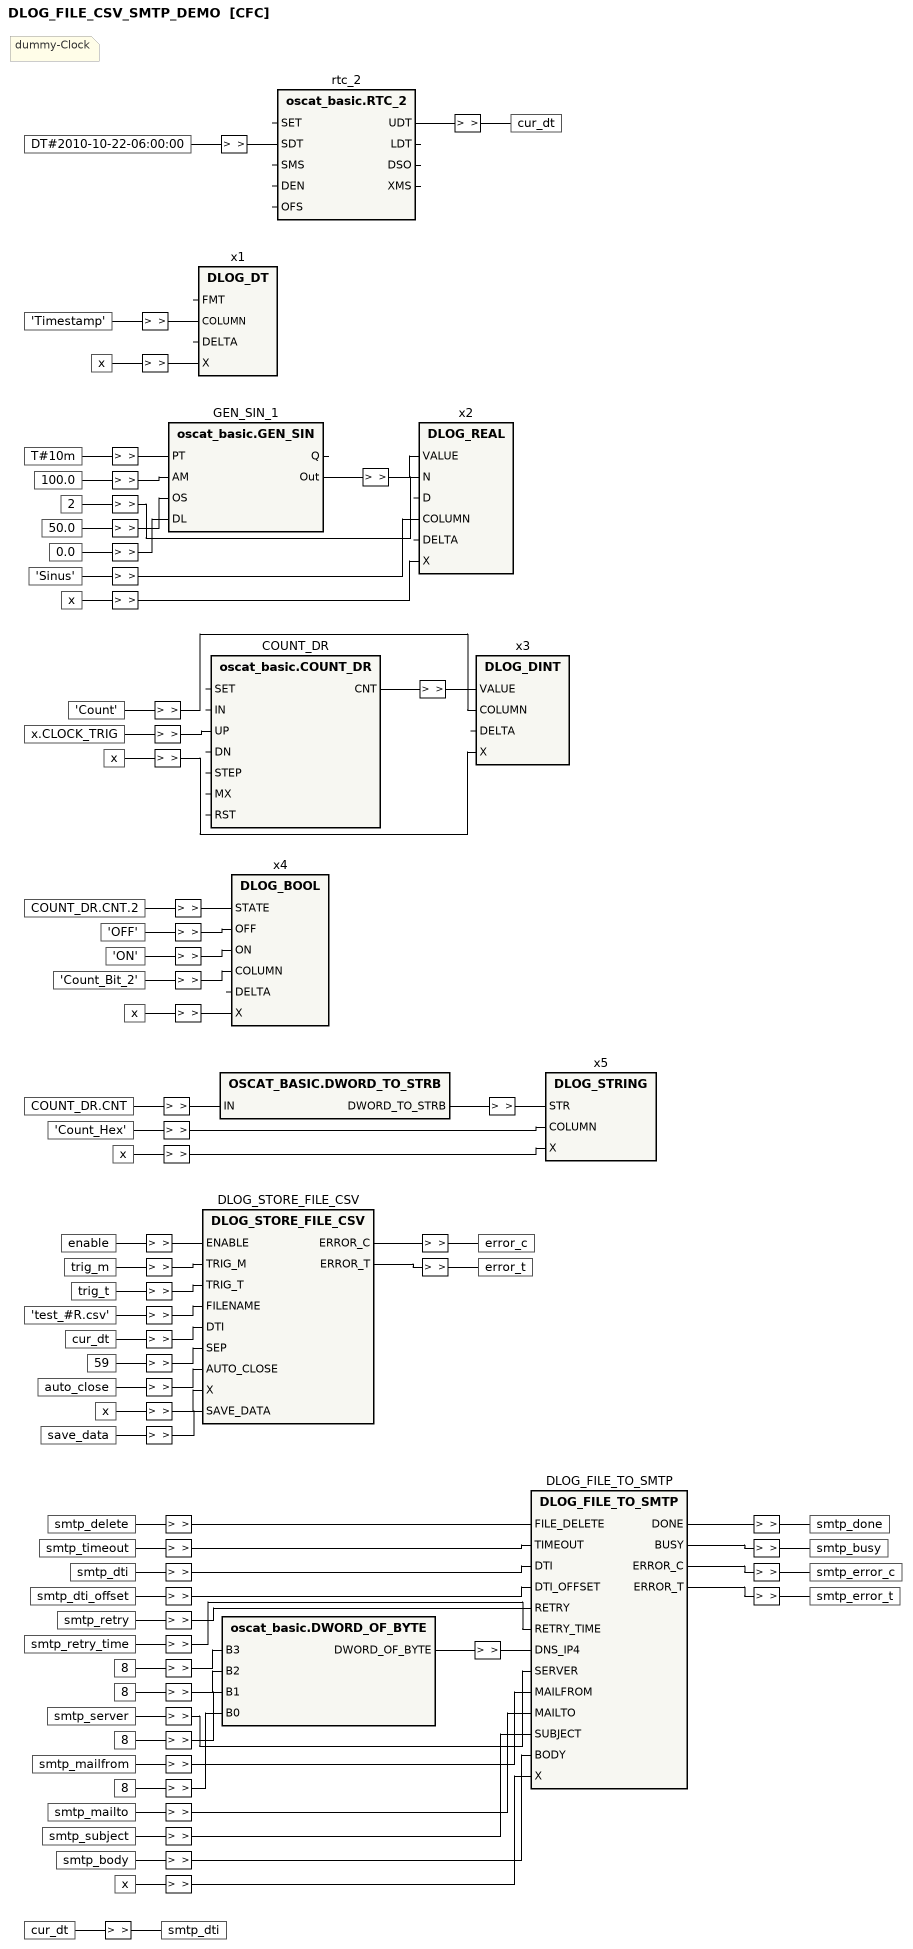
(* CFC diagram, written out as Structured Text *)
(* dummy-Clock *)
rtc_2(SDT := DT#2010-10-22-06:00:00);
cur_dt := rtc_2.UDT;
x1(COLUMN := 'Timestamp', X := x);
GEN_SIN_1(PT := T#10m, AM := 100.0, OS := 50.0, DL := 0.0);
x2(VALUE := GEN_SIN_1.Out, N := 2, COLUMN := 'Sinus', X := x);
COUNT_DR(UP := x.CLOCK_TRIG);
x3(VALUE := COUNT_DR.CNT, COLUMN := 'Count', X := x);
x4(STATE := COUNT_DR.CNT.2, OFF := 'OFF', ON := 'ON', COLUMN := 'Count_Bit_2', X := x);
x5(STR := OSCAT_BASIC.DWORD_TO_STRB(COUNT_DR.CNT), COLUMN := 'Count_Hex', X := x);
DLOG_STORE_FILE_CSV(ENABLE := enable, TRIG_M := trig_m, TRIG_T := trig_t, FILENAME := 'test_#R.csv', DTI := cur_dt, SEP := 59, AUTO_CLOSE := auto_close, X := x, SAVE_DATA := save_data);
error_c := DLOG_STORE_FILE_CSV.ERROR_C;
error_t := DLOG_STORE_FILE_CSV.ERROR_T;
DLOG_FILE_TO_SMTP(FILE_DELETE := smtp_delete, TIMEOUT := smtp_timeout, DTI := smtp_dti, DTI_OFFSET := smtp_dti_offset, RETRY := smtp_retry, RETRY_TIME := smtp_retry_time, DNS_IP4 := oscat_basic.DWORD_OF_BYTE(8, 8, 8, 8), SERVER := smtp_server, MAILFROM := smtp_mailfrom, MAILTO := smtp_mailto, SUBJECT := smtp_subject, BODY := smtp_body, X := x);
smtp_done := DLOG_FILE_TO_SMTP.DONE;
smtp_busy := DLOG_FILE_TO_SMTP.BUSY;
smtp_error_c := DLOG_FILE_TO_SMTP.ERROR_C;
smtp_error_t := DLOG_FILE_TO_SMTP.ERROR_T;
smtp_dti := cur_dt;
END_PROGRAM

PROGRAM DLOG_FILE_HTML_DEMO
  VAR
    cur_dt : DT;
    enable : BOOL := TRUE;
    trig_t : TIME := TIME#5s0ms;
    trig_m : BOOL;
    error_c : DWORD;
    error_t : BYTE;
    auto_close : TIME := TIME#10s0ms;
    x1 : DLOG_DT;
    x2 : DLOG_REAL;
    x3 : DLOG_DINT;
    x4 : DLOG_BOOL;
    x5 : DLOG_STRING;
    x : DLOG_DATA;
    RTC_2 : oscat_basic.RTC_2;
    DLOG_STORE_FILE_HTML : DLOG_STORE_FILE_HTML;
    GEN_SIN_1 : oscat_basic.GEN_SIN;
    COUNT_DR : oscat_basic.COUNT_DR;
    html_caption : STRING := 'Das ist der Titel';
    html_tr_even : STRING := 'BGCOLOR=#B3B7FF';
    html_tr_odd : STRING := 'BGCOLOR=#E0E0E0';
    html_tr_head : STRING := 'BGCOLOR=#FFFF40';
    html_table : STRING := 'BORDER="1"';
  END_VAR
  VAR RETAIN
    save_data : DLOG_SAVE;
  END_VAR

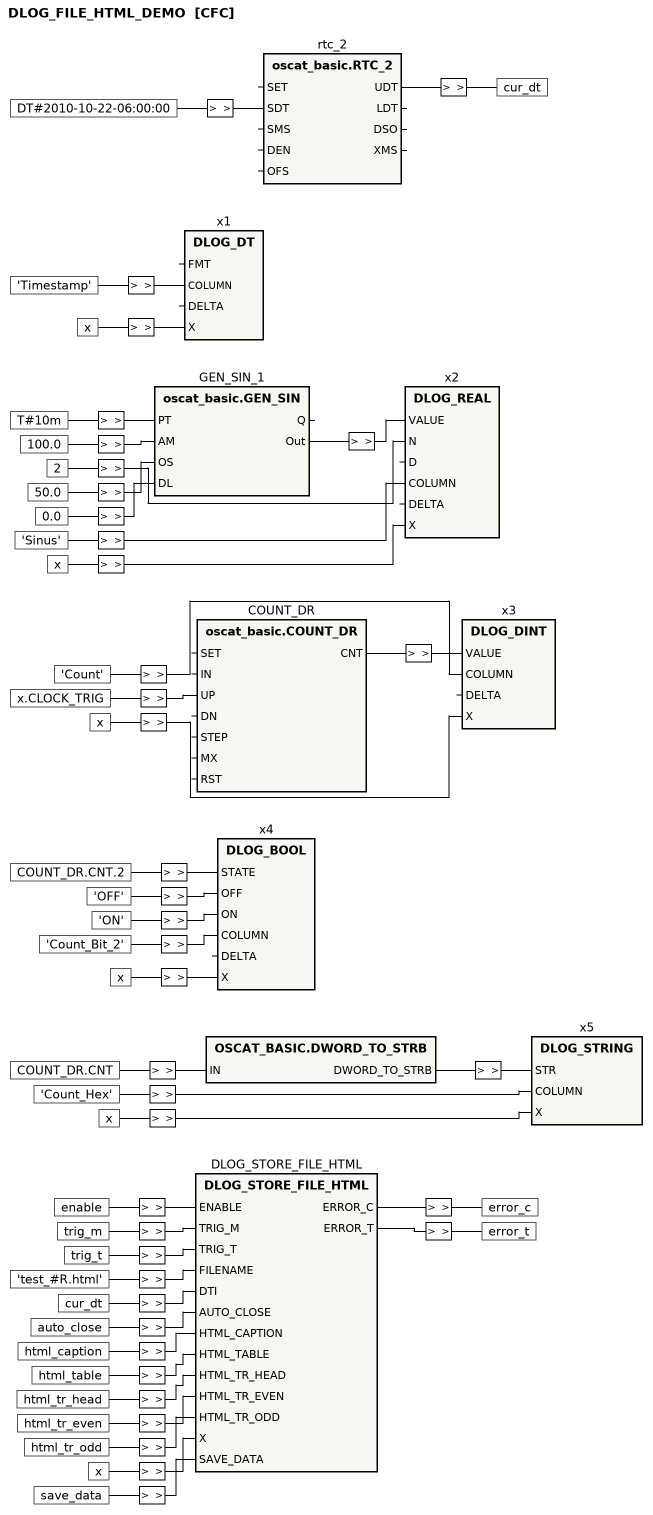
(* CFC diagram, written out as Structured Text *)
rtc_2(SDT := DT#2010-10-22-06:00:00);
cur_dt := rtc_2.UDT;
x1(COLUMN := 'Timestamp', X := x);
GEN_SIN_1(PT := T#10m, AM := 100.0, OS := 50.0, DL := 0.0);
x2(VALUE := GEN_SIN_1.Out, N := 2, COLUMN := 'Sinus', X := x);
COUNT_DR(UP := x.CLOCK_TRIG);
x3(VALUE := COUNT_DR.CNT, COLUMN := 'Count', X := x);
x4(STATE := COUNT_DR.CNT.2, OFF := 'OFF', ON := 'ON', COLUMN := 'Count_Bit_2', X := x);
x5(STR := OSCAT_BASIC.DWORD_TO_STRB(COUNT_DR.CNT), COLUMN := 'Count_Hex', X := x);
DLOG_STORE_FILE_HTML(ENABLE := enable, TRIG_M := trig_m, TRIG_T := trig_t, FILENAME := 'test_#R.html', DTI := cur_dt, AUTO_CLOSE := auto_close, HTML_CAPTION := html_caption, HTML_TABLE := html_table, HTML_TR_HEAD := html_tr_head, HTML_TR_EVEN := html_tr_even, HTML_TR_ODD := html_tr_odd, X := x, SAVE_DATA := save_data);
error_c := DLOG_STORE_FILE_HTML.ERROR_C;
error_t := DLOG_STORE_FILE_HTML.ERROR_T;
END_PROGRAM

PROGRAM DLOG_FILE_XML_DEMO
  VAR
    cur_dt : DT;
    enable : BOOL := TRUE;
    trig_t : TIME := TIME#5s0ms;
    trig_m : BOOL;
    error_c : DWORD;
    error_t : BYTE;
    auto_close : TIME := TIME#10s0ms;
    x1 : DLOG_DT;
    x2 : DLOG_REAL;
    x3 : DLOG_DINT;
    x4 : DLOG_BOOL;
    x5 : DLOG_STRING;
    x : DLOG_DATA;
    RTC_2 : oscat_basic.RTC_2;
    DLOG_STORE_FILE_XML : DLOG_STORE_FILE_XML;
    GEN_SIN_1 : oscat_basic.GEN_SIN;
    COUNT_DR : oscat_basic.COUNT_DR;
  END_VAR
  VAR RETAIN
    save_data : DLOG_SAVE;
  END_VAR

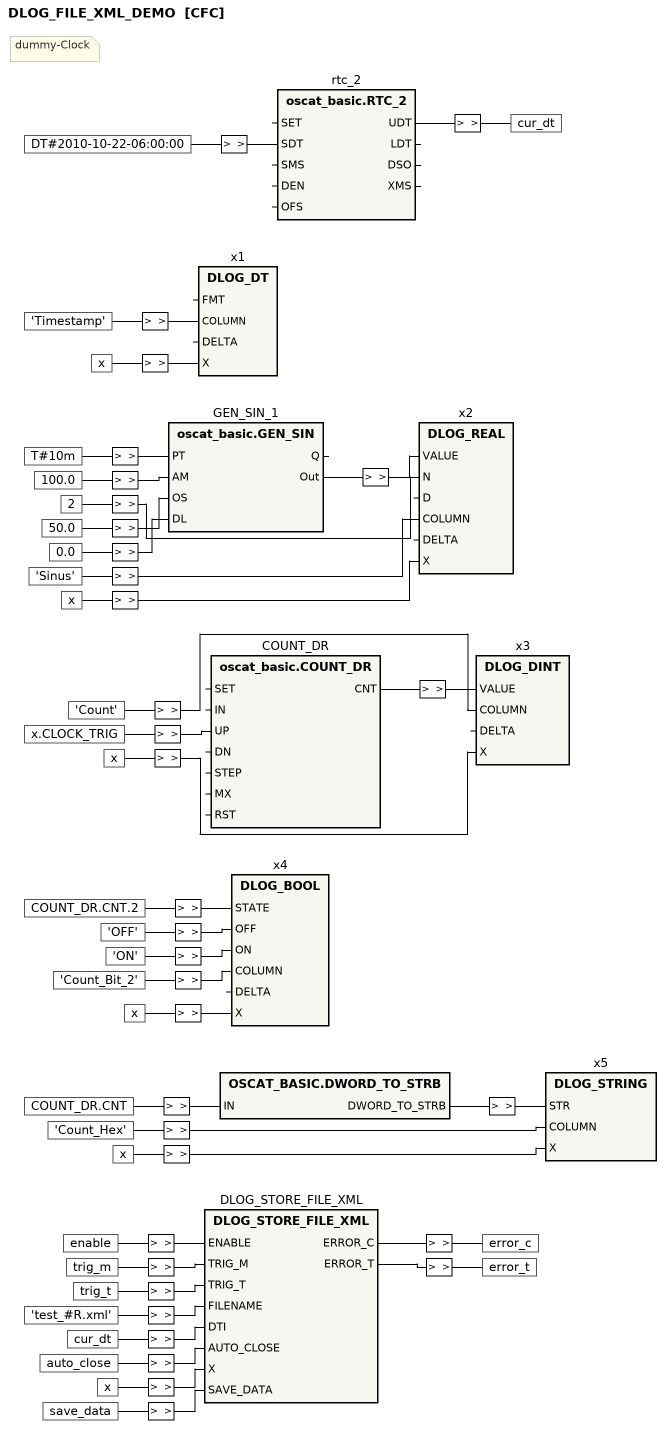
(* CFC diagram, written out as Structured Text *)
(* dummy-Clock *)
rtc_2(SDT := DT#2010-10-22-06:00:00);
cur_dt := rtc_2.UDT;
x1(COLUMN := 'Timestamp', X := x);
GEN_SIN_1(PT := T#10m, AM := 100.0, OS := 50.0, DL := 0.0);
x2(VALUE := GEN_SIN_1.Out, N := 2, COLUMN := 'Sinus', X := x);
COUNT_DR(UP := x.CLOCK_TRIG);
x3(VALUE := COUNT_DR.CNT, COLUMN := 'Count', X := x);
x4(STATE := COUNT_DR.CNT.2, OFF := 'OFF', ON := 'ON', COLUMN := 'Count_Bit_2', X := x);
x5(STR := OSCAT_BASIC.DWORD_TO_STRB(COUNT_DR.CNT), COLUMN := 'Count_Hex', X := x);
DLOG_STORE_FILE_XML(ENABLE := enable, TRIG_M := trig_m, TRIG_T := trig_t, FILENAME := 'test_#R.xml', DTI := cur_dt, AUTO_CLOSE := auto_close, X := x, SAVE_DATA := save_data);
error_c := DLOG_STORE_FILE_XML.ERROR_C;
error_t := DLOG_STORE_FILE_XML.ERROR_T;
END_PROGRAM

PROGRAM DLOG_MYSQL_DEMO
  VAR
    cur_dt : DT;
    enable : BOOL := TRUE;
    trig_t : TIME := TIME#5s0ms;
    trig_m : BOOL;
    error_c : DWORD;
    error_t : BYTE;
    x1 : DLOG_DT;
    x2 : DLOG_REAL;
    x3 : DLOG_DINT;
    x4 : DLOG_BOOL;
    x5 : DLOG_STRING;
    x : DLOG_DATA;
    mysql_info : MYSQL_INFO;
    RTC_2 : oscat_basic.RTC_2;
    GEN_SIN_1 : oscat_basic.GEN_SIN;
    COUNT_DR : oscat_basic.COUNT_DR;
    DLOG_STORE_MYSQL : DLOG_STORE_MYSQL;
    url : STRING(OSCAT_BASIC.STRING_LENGTH) := 'myuser:mypassword@192.168.178.21';  (* url : STRING := 'myuser:mypassword@127.0.0.1'; *)
    db_name : STRING(64) := 'oscat_db';
    tb_name : STRING(64) := 'oscat_tb';
    auto_delete : UDINT := 0;
    timeout : TIME := TIME#10s0ms;
  END_VAR

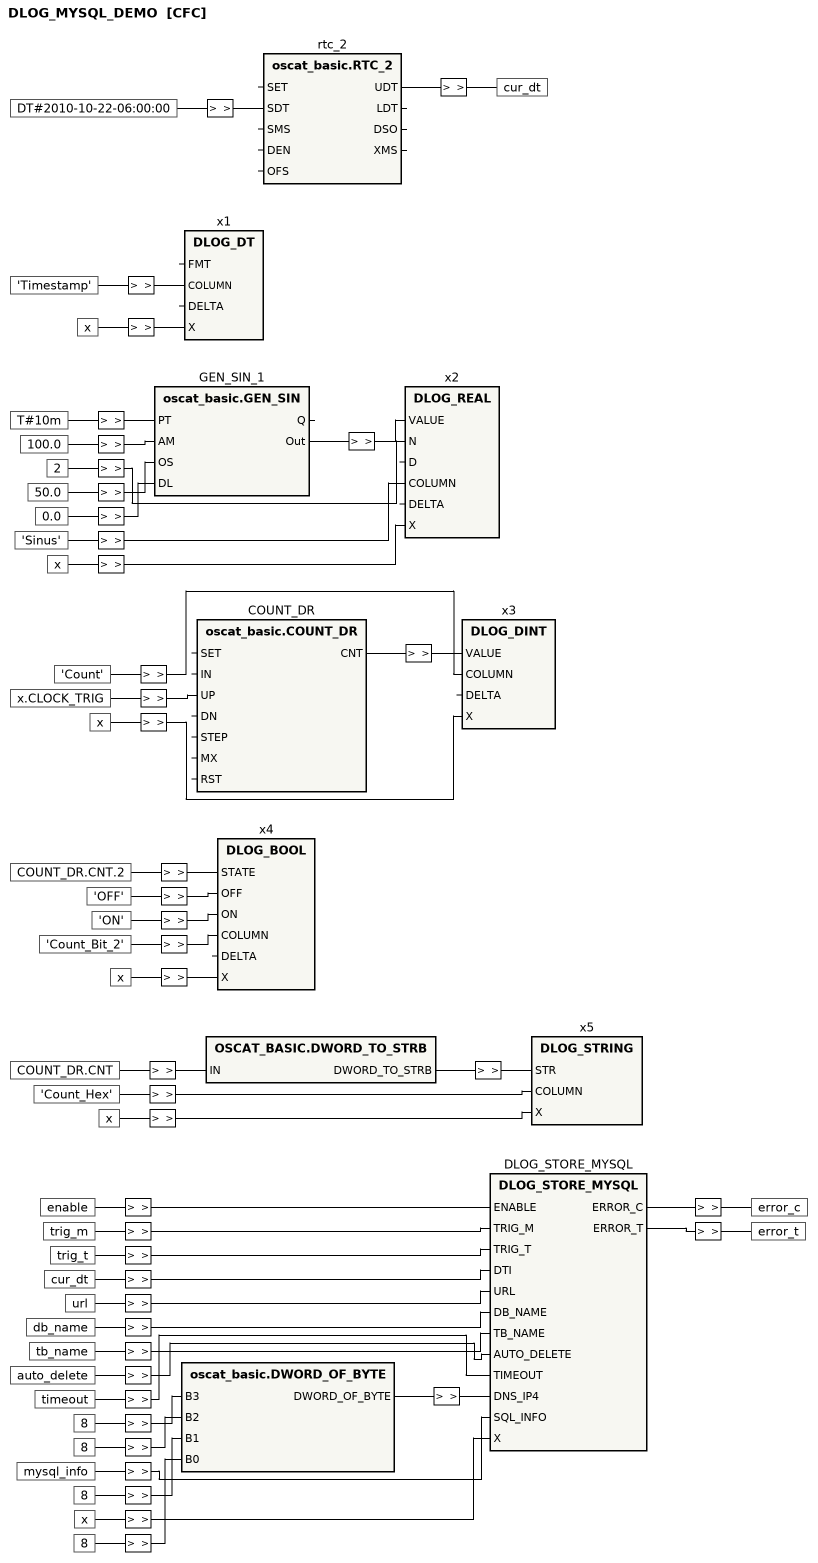
(* CFC diagram, written out as Structured Text *)
rtc_2(SDT := DT#2010-10-22-06:00:00);
cur_dt := rtc_2.UDT;
x1(COLUMN := 'Timestamp', X := x);
GEN_SIN_1(PT := T#10m, AM := 100.0, OS := 50.0, DL := 0.0);
x2(VALUE := GEN_SIN_1.Out, N := 2, COLUMN := 'Sinus', X := x);
COUNT_DR(UP := x.CLOCK_TRIG);
x3(VALUE := COUNT_DR.CNT, COLUMN := 'Count', X := x);
x4(STATE := COUNT_DR.CNT.2, OFF := 'OFF', ON := 'ON', COLUMN := 'Count_Bit_2', X := x);
x5(STR := OSCAT_BASIC.DWORD_TO_STRB(COUNT_DR.CNT), COLUMN := 'Count_Hex', X := x);
DLOG_STORE_MYSQL(ENABLE := enable, TRIG_M := trig_m, TRIG_T := trig_t, DTI := cur_dt, URL := url, DB_NAME := db_name, TB_NAME := tb_name, AUTO_DELETE := auto_delete, TIMEOUT := timeout, DNS_IP4 := oscat_basic.DWORD_OF_BYTE(8, 8, 8, 8), SQL_INFO := mysql_info, X := x);
error_t := DLOG_STORE_MYSQL.ERROR_T;
error_c := DLOG_STORE_MYSQL.ERROR_C;
END_PROGRAM

PROGRAM DLOG_RRD_DEMO
  VAR
    cur_dt : DT;
    trig_t : TIME := TIME#50s0ms;
    trig_m : BOOL;
    rrd_error_c : DWORD;
    rrd_error_t : BYTE;
    rrd_enable : BOOL := TRUE;
    rrd_url : STRING(OSCAT_BASIC.STRING_LENGTH) := '192.168.178.21/rrd/test_rrd2.php?rrd_db=test.rrd&value=';  (* rrd_url : STRING(OSCAT_BASIC.STRING_LENGTH) := 'http://xxx.com/myhouse/rrd/test_rrd.php?rrd_db=test.rrd&value='; *)
    rrd_timeout : TIME := TIME#5s0ms;
    RTC_2 : oscat_basic.RTC_2;
    DLOG_STORE_RRD : DLOG_STORE_RRD;
    x : DLOG_DATA;
    x1 : DLOG_DINT;
    x2 : DLOG_DINT;
    x3 : DLOG_REAL;
    x4 : DLOG_REAL;
    x5 : DLOG_REAL;
    x6 : DLOG_REAL;
    x7 : DLOG_REAL;
    GEN_SIN_1 : oscat_basic.GEN_SIN;
    GEN_SIN_2 : oscat_basic.GEN_SIN;
    GEN_SIN_3 : oscat_basic.GEN_SIN;
    GEN_RMP_1 : oscat_basic.GEN_RMP;
    GEN_RMP_2 : oscat_basic.GEN_RMP;
  END_VAR

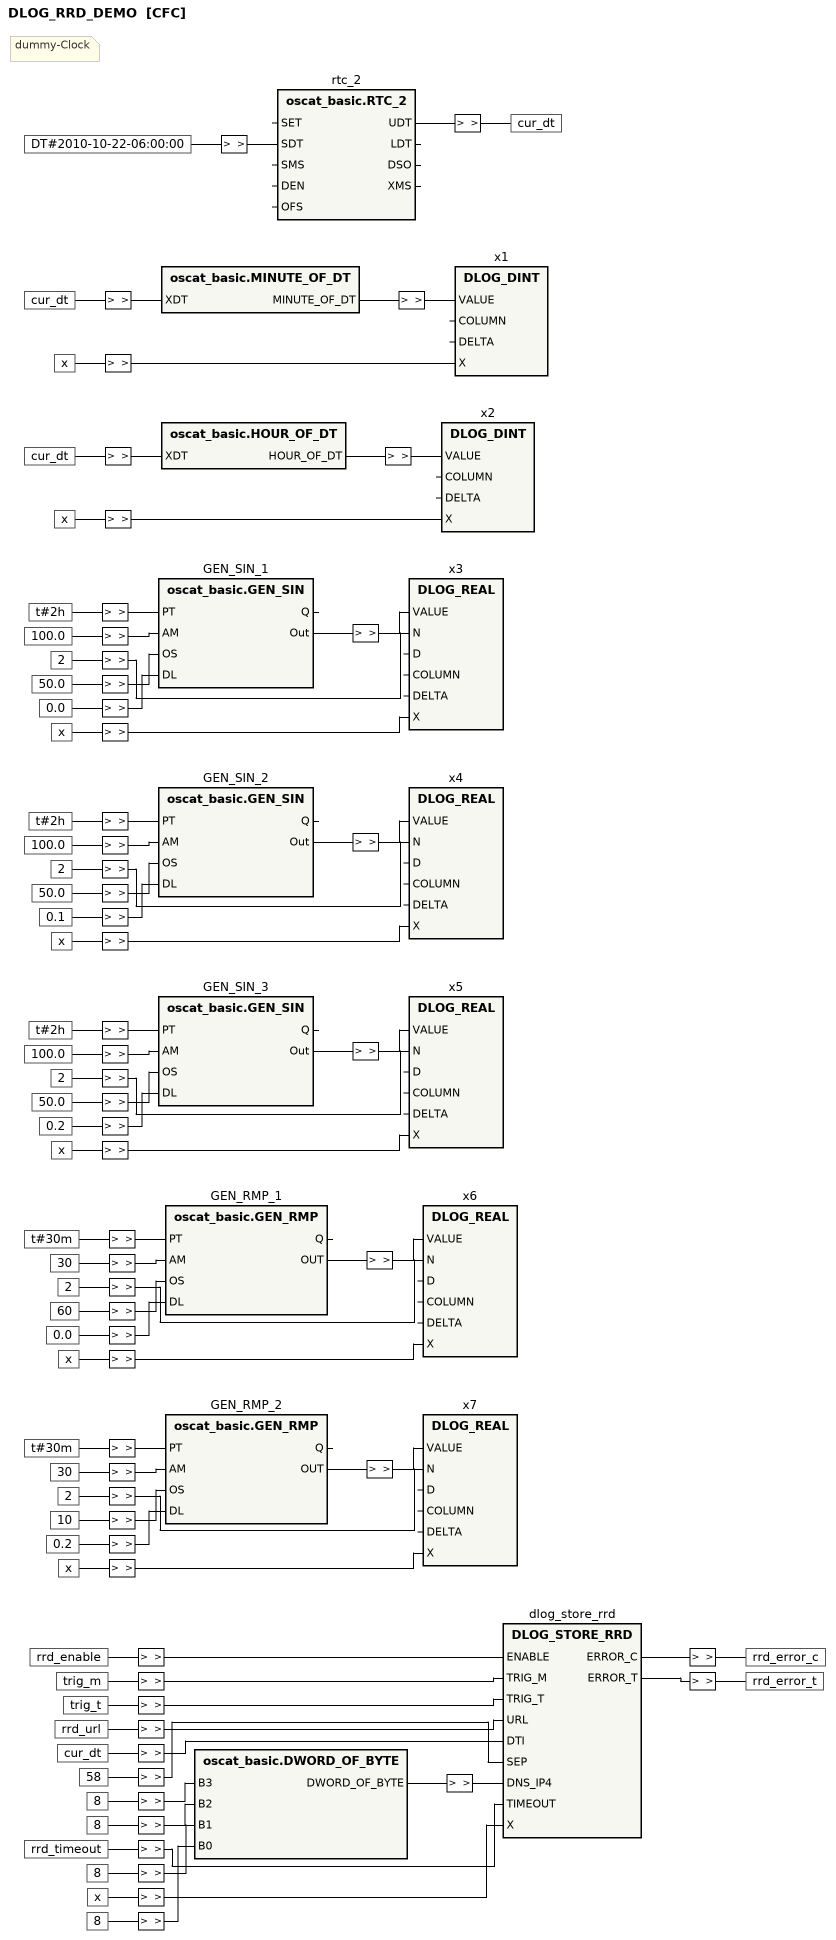
(* CFC diagram, written out as Structured Text *)
(* dummy-Clock *)
rtc_2(SDT := DT#2010-10-22-06:00:00);
cur_dt := rtc_2.UDT;
x1(VALUE := oscat_basic.MINUTE_OF_DT(cur_dt), X := x);
x2(VALUE := oscat_basic.HOUR_OF_DT(cur_dt), X := x);
GEN_SIN_1(PT := t#2h, AM := 100.0, OS := 50.0, DL := 0.0);
x3(VALUE := GEN_SIN_1.Out, N := 2, X := x);
GEN_SIN_2(PT := t#2h, AM := 100.0, OS := 50.0, DL := 0.1);
x4(VALUE := GEN_SIN_2.Out, N := 2, X := x);
GEN_SIN_3(PT := t#2h, AM := 100.0, OS := 50.0, DL := 0.2);
x5(VALUE := GEN_SIN_3.Out, N := 2, X := x);
GEN_RMP_1(PT := t#30m, AM := 30, OS := 60, DL := 0.0);
x6(VALUE := GEN_RMP_1.OUT, N := 2, X := x);
GEN_RMP_2(PT := t#30m, AM := 30, OS := 10, DL := 0.2);
x7(VALUE := GEN_RMP_2.OUT, N := 2, X := x);
dlog_store_rrd(ENABLE := rrd_enable, TRIG_M := trig_m, TRIG_T := trig_t, URL := rrd_url, DTI := cur_dt, SEP := 58, DNS_IP4 := oscat_basic.DWORD_OF_BYTE(8, 8, 8, 8), TIMEOUT := rrd_timeout, X := x);
rrd_error_c := dlog_store_rrd.ERROR_C;
rrd_error_t := dlog_store_rrd.ERROR_T;
END_PROGRAM

PROGRAM DNS_DYN_DEMO
  VAR
    DNS_DYN : DNS_DYN;
    IP_C : IP_C;
    S_BUF : NETWORK_BUFFER;
    R_BUF : NETWORK_BUFFER;
    IP_CONTROL : IP_CONTROL;
    enable : BOOL;
    done : BOOL;
    error_c : DWORD;
    error_t : BYTE;
    busy : BOOL;
    COUNT_DR : oscat_basic.COUNT_DR;
    z : DWORD;
    GET_WAN_IP : GET_WAN_IP;
    t1 : TON;
    done2 : BOOL;
    error_c2 : DWORD;
    error_t2 : BYTE;
    update : BOOL;
    new_ip : BOOL;
    wan_ip4 : DWORD;
  END_VAR

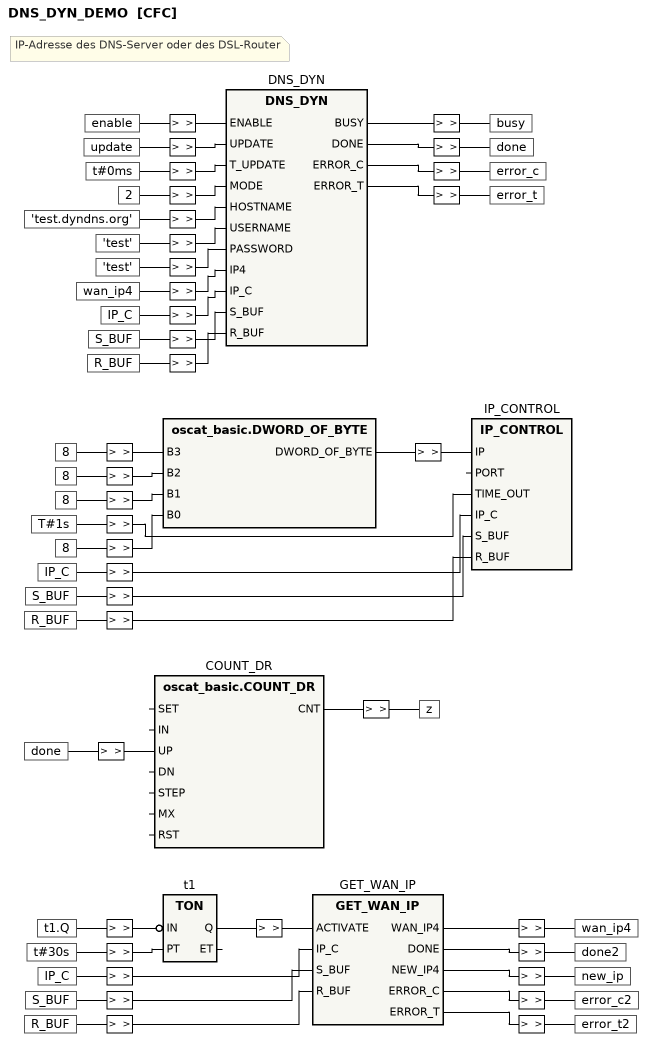
(* CFC diagram, written out as Structured Text *)
DNS_DYN(ENABLE := enable, UPDATE := update, T_UPDATE := t#0ms, MODE := 2, HOSTNAME := 'test.dyndns.org', USERNAME := 'test', PASSWORD := 'test', IP4 := wan_ip4, IP_C := IP_C, S_BUF := S_BUF, R_BUF := R_BUF);
busy := DNS_DYN.BUSY;
done := DNS_DYN.DONE;
error_c := DNS_DYN.ERROR_C;
error_t := DNS_DYN.ERROR_T;
(* IP-Adresse des DNS-Server oder des DSL-Router *)
IP_CONTROL(IP := oscat_basic.DWORD_OF_BYTE(8, 8, 8, 8), TIME_OUT := T#1s, IP_C := IP_C, S_BUF := S_BUF, R_BUF := R_BUF);
COUNT_DR(UP := done);
z := COUNT_DR.CNT;
wan_ip4 := GET_WAN_IP.WAN_IP4;
t1(IN := NOT t1.Q, PT := t#30s);
GET_WAN_IP(ACTIVATE := t1.Q, IP_C := IP_C, S_BUF := S_BUF, R_BUF := R_BUF);
done2 := GET_WAN_IP.DONE;
new_ip := GET_WAN_IP.NEW_IP4;
error_c2 := GET_WAN_IP.ERROR_C;
error_t2 := GET_WAN_IP.ERROR_T;
END_PROGRAM

PROGRAM DNS_REV_DEMO
  VAR
    DNS_REV_CLIENT : DNS_REV_CLIENT;
    IP_C : IP_C;
    S_BUF : NETWORK_BUFFER;
    R_BUF : NETWORK_BUFFER;
    IP_CONTROL : IP_CONTROL;
    activate : BOOL := TRUE;
    done : BOOL;
    error : DWORD;
    domain : STRING;
  END_VAR

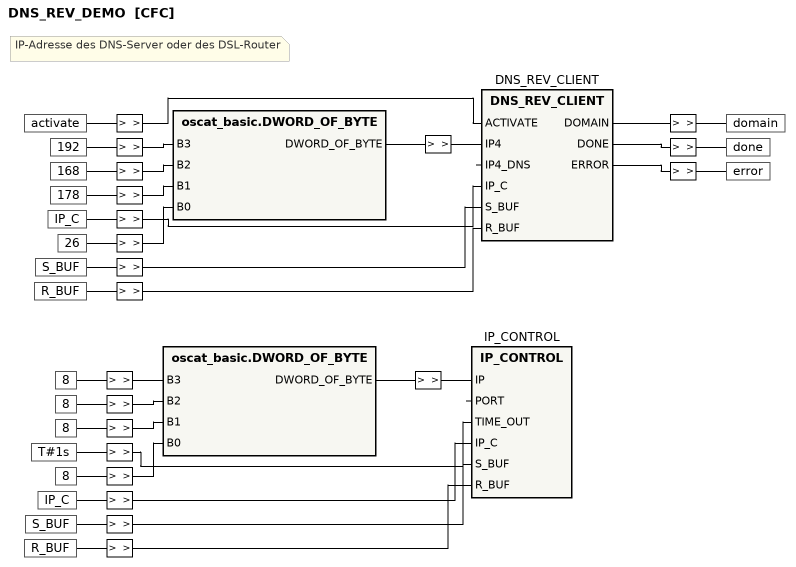
(* CFC diagram, written out as Structured Text *)
DNS_REV_CLIENT(ACTIVATE := activate, IP4 := oscat_basic.DWORD_OF_BYTE(192, 168, 178, 26), IP_C := IP_C, S_BUF := S_BUF, R_BUF := R_BUF);
domain := DNS_REV_CLIENT.DOMAIN;
done := DNS_REV_CLIENT.DONE;
error := DNS_REV_CLIENT.ERROR;
(* IP-Adresse des DNS-Server oder des DSL-Router *)
IP_CONTROL(IP := oscat_basic.DWORD_OF_BYTE(8, 8, 8, 8), TIME_OUT := T#1s, IP_C := IP_C, S_BUF := S_BUF, R_BUF := R_BUF);
END_PROGRAM

PROGRAM DNS_SNTP_SYSLOG_DEMO
  VAR
    IP_C : IP_C;
    S_BUF : NETWORK_BUFFER;
    R_BUF : NETWORK_BUFFER;
    IP_CONTROL_1 : IP_CONTROL;
    DNS_CLIENT : DNS_CLIENT;
    SNTP_CLIENT : SNTP_CLIENT;
    SNTP_SERVER : SNTP_SERVER;
    COUNT_DR : oscat_basic.COUNT_DR;
    RTC_2 : oscat_basic.RTC_2;
    count_cycles : DWORD;
    dns_error : DWORD;
    sntp_error : DWORD;
    freigabe : BOOL;
    dso : BOOL;
    xms : INT;
    sntp_srv_enable : BOOL;
    cur_UDT : DT;
    SYS_LOG : SYS_LOG;
    sys_log_option : BYTE := 2#100;
    TON_1 : TON;
    tp_sys_log : BOOL;
    error_sys_log : DWORD;
    sys_time : TIME;
    cur_LOCAL_DT : DT;
  END_VAR

(* CFC diagram, written out as Structured Text *)
TON_1(IN := NOT TON_1.Q, PT := T#10s);
freigabe := TON_1.Q;
sys_time := TON_1.ET;
DNS_CLIENT(ACTIVATE := freigabe, DOMAIN := 'time.windows.com', IP_C := IP_C, S_BUF := S_BUF, R_BUF := R_BUF);
dns_error := DNS_CLIENT.ERROR;
SNTP_CLIENT(IP4 := DNS_CLIENT.IP4, ACTIVATE := DNS_CLIENT.DONE, IP_C := IP_C, S_BUF := S_BUF, R_BUF := R_BUF);
sntp_error := SNTP_CLIENT.ERROR;
RTC_2(SET := SNTP_CLIENT.DONE_P, SDT := SNTP_CLIENT.UDT, SMS := SNTP_CLIENT.XMS, DEN := TRUE, OFS := 1);
cur_UDT := RTC_2.UDT;
cur_LOCAL_DT := RTC_2.LOCAL_DT;
dso := RTC_2.DSO;
xms := RTC_2.XMS;
SNTP_SERVER(ENABLE := sntp_srv_enable, UDT := cur_UDT, XMS := xms, IP_C := IP_C, S_BUF := S_BUF, R_BUF := R_BUF);
COUNT_DR(UP := freigabe, MX := DWORD#16#FFFFFFFF);
count_cycles := COUNT_DR.CNT;
(* IP-Adresse des DNS-Server oder des DSL-Router *)
IP_CONTROL_1(IP := oscat_basic.DWORD_OF_BYTE(8, 8, 8, 8), TIME_OUT := T#4s, IP_C := IP_C, S_BUF := S_BUF, R_BUF := R_BUF);
SYS_LOG(ACTIVATE := freigabe, LOC_DT := cur_LOCAL_DT, SERVER_IP4 := oscat_basic.DWORD_OF_BYTE(192, 168, 178, 26), FACILITY := 2, SEVERITY := 3, TAG := 'SyslogGEN', HOSTNAME := 'privat-str', MESSAGE := 'This is a test message generated by OSCAT SYSLOG', OPTION := sys_log_option, IP_C := IP_C, S_BUF := S_BUF, R_BUF := R_BUF);
tp_sys_log := SYS_LOG.DONE_P;
error_sys_log := SYS_LOG.ERROR;
END_PROGRAM

PROGRAM FILE_BLOCK_DEMO
  VAR
    PT : NETWORK_BUFFER;
    fsd : FILE_SERVER_DATA;
    FILE_SERVER : FILE_SERVER;
    FILE_BLOCK : FILE_BLOCK;
    filename : STRING := 'config.ini';
    data : BYTE;
    error : BYTE;
    mode : BYTE;
    pos : UDINT;
  END_VAR

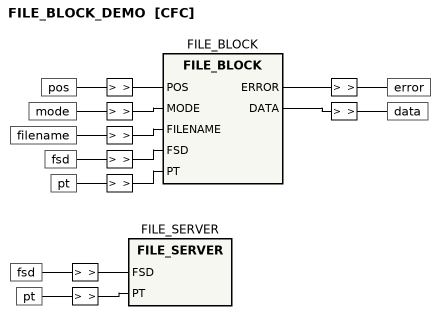
(* CFC diagram, written out as Structured Text *)
FILE_BLOCK(POS := pos, MODE := mode, FILENAME := filename, FSD := fsd, PT := pt);
error := FILE_BLOCK.ERROR;
data := FILE_BLOCK.DATA;
FILE_SERVER(FSD := fsd, PT := pt);
END_PROGRAM

PROGRAM FTP_CLIENT_DEMO
  VAR
    FTP_CLIENT : FTP_CLIENT;
    ftp_activate : BOOL;
    ftp_done : BOOL;
    ftp_busy : BOOL;
    ftp_error_c : DWORD;
    ftp_error_t : BYTE;
    ftp_url : STRING := 'ftp://581920:123456@oscat.atwebpages.com:2000/subordner/';
    ftp_filename : STRING := '0100kb.bin';
    ftp_download : BOOL := TRUE;
    ftp_activ : BOOL := FALSE;
    file_delete : BOOL := FALSE;
    ftp_timeout : TIME := TIME#30s0ms;
    zeit : TIME := TIME#30s0ms;
    stop : BOOL;
    start : BOOL := TRUE;
    reset : BOOL;
    error : DWORD;
    ok : DWORD;
    CLK_PRG_1 : oscat_basic.CLK_PRG;
    COUNT_DR_1 : oscat_basic.COUNT_DR;
    COUNT_DR_2 : oscat_basic.COUNT_DR;
  END_VAR
  VAR  (* added by the conversion: wires and edge detectors of the diagram *)
    _oscat_basic_DWORD_OF_BYTE16_OUT : ANY;
    _oscat_basic_DWORD_OF_BYTE26_OUT : ANY;
    _AND46_OUT : BOOL;
  END_VAR

(* CFC diagram, written out as Structured Text *)
ftp_client(ACTIVATE := ftp_activate, FILENAME := ftp_filename, FTP_URL := ftp_url, FTP_DOWNLOAD := ftp_download, FTP_ACTIV := ftp_activ, FILE_DELETE := file_delete, TIMEOUT := ftp_timeout, DNS_IP4 := _oscat_basic_DWORD_OF_BYTE16_OUT, PLC_IP4 := _oscat_basic_DWORD_OF_BYTE26_OUT);
ftp_done := ftp_client.DONE;
ftp_busy := ftp_client.BUSY;
ftp_error_c := ftp_client.ERROR_C;
ftp_error_t := ftp_client.ERROR_T;
CLK_PRG_1(PT := zeit);
_AND46_OUT := CLK_PRG_1.Q AND NOT stop AND start;
ftp_activate := _AND46_OUT OR reset;
stop := ftp_error_t <> 0;
COUNT_DR_1(UP := stop);
error := COUNT_DR_1.CNT;
COUNT_DR_2(UP := ftp_done);
ok := COUNT_DR_2.CNT;
_oscat_basic_DWORD_OF_BYTE16_OUT := oscat_basic.DWORD_OF_BYTE(8, 8, 8, 8);
_oscat_basic_DWORD_OF_BYTE26_OUT := oscat_basic.DWORD_OF_BYTE(192, 168, 178, 25);
END_PROGRAM

PROGRAM GET_WAN_IP_DEMO
  VAR
    GET_WAN_IP : GET_WAN_IP;
    IP_C : IP_C;
    S_BUF : NETWORK_BUFFER;
    R_BUF : NETWORK_BUFFER;
    IP_CONTROL_1 : IP_CONTROL;
    activate : BOOL;
    done : BOOL;
    error_c : DWORD;
    error_t : BYTE;
    wan_ip : STRING;
    new_ip : BOOL;
  END_VAR

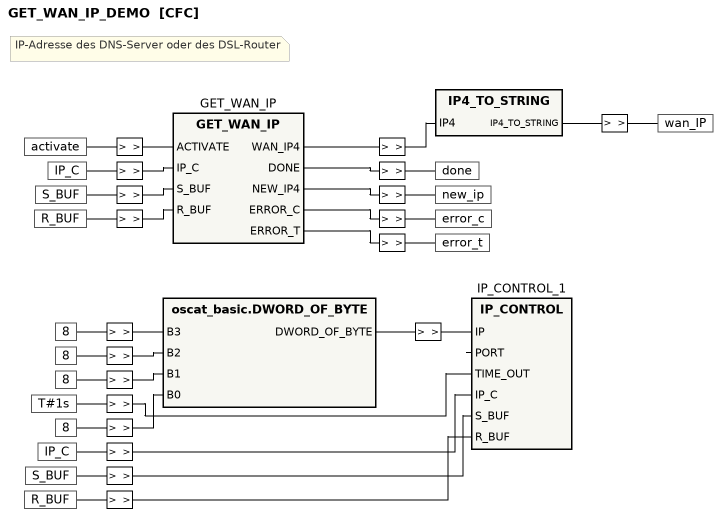
(* CFC diagram, written out as Structured Text *)
GET_WAN_IP(ACTIVATE := activate, IP_C := IP_C, S_BUF := S_BUF, R_BUF := R_BUF);
done := GET_WAN_IP.DONE;
new_ip := GET_WAN_IP.NEW_IP4;
error_c := GET_WAN_IP.ERROR_C;
(* IP-Adresse des DNS-Server oder des DSL-Router *)
error_t := GET_WAN_IP.ERROR_T;
wan_IP := IP4_TO_STRING(GET_WAN_IP.WAN_IP4);
IP_CONTROL_1(IP := oscat_basic.DWORD_OF_BYTE(8, 8, 8, 8), TIME_OUT := T#1s, IP_C := IP_C, S_BUF := S_BUF, R_BUF := R_BUF);
END_PROGRAM

PROGRAM HTTP_DEMO
  VAR
    url_text : STRING := 'http://weather.yahooapis.com/forecastrss?p=94089&u=c';
    URL_DATA : URL;
    IP_C : IP_C;
    S_BUF : NETWORK_BUFFER;
    R_BUF : NETWORK_BUFFER;
    IP_CONTROL_1 : IP_CONTROL;
    DNS_CLIENT : DNS_CLIENT;
    HTTP_GET : HTTP_GET;
    http_release : BOOL;
    enable : BOOL := TRUE;
    http_status : STRING;
    header_start : UINT;
    header_stop : UINT;
    body_start : UINT;
    body_stop : UINT;
    http_get_done : BOOL;
    http_get_error : DWORD;
    COUNT_DR : OSCAT_BASIC.COUNT_DR;
    cycles : DWORD;
    TON_1 : TON;
    F_TRIG : F_TRIG;
  END_VAR

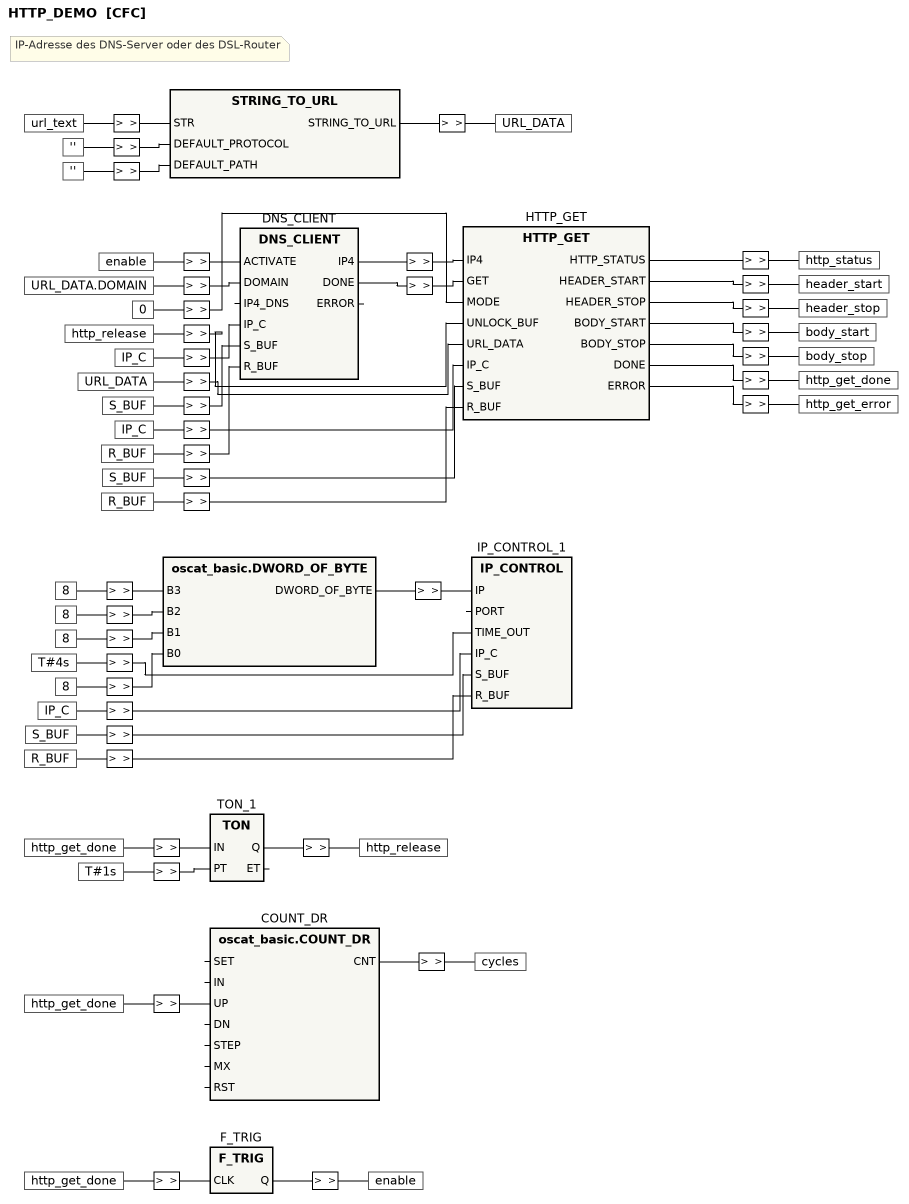
(* CFC diagram, written out as Structured Text *)
URL_DATA := STRING_TO_URL(url_text, '', '');
DNS_CLIENT(ACTIVATE := enable, DOMAIN := URL_DATA.DOMAIN, IP_C := IP_C, S_BUF := S_BUF, R_BUF := R_BUF);
HTTP_GET(IP4 := DNS_CLIENT.IP4, GET := DNS_CLIENT.DONE, MODE := 0, UNLOCK_BUF := http_release, URL_DATA := URL_DATA, IP_C := IP_C, S_BUF := S_BUF, R_BUF := R_BUF);
http_status := HTTP_GET.HTTP_STATUS;
header_start := HTTP_GET.HEADER_START;
header_stop := HTTP_GET.HEADER_STOP;
body_start := HTTP_GET.BODY_START;
body_stop := HTTP_GET.BODY_STOP;
http_get_done := HTTP_GET.DONE;
http_get_error := HTTP_GET.ERROR;
(* IP-Adresse des DNS-Server oder des DSL-Router *)
IP_CONTROL_1(IP := oscat_basic.DWORD_OF_BYTE(8, 8, 8, 8), TIME_OUT := T#4s, IP_C := IP_C, S_BUF := S_BUF, R_BUF := R_BUF);
TON_1(IN := http_get_done, PT := T#1s);
http_release := TON_1.Q;
COUNT_DR(UP := http_get_done);
cycles := COUNT_DR.CNT;
F_TRIG(CLK := http_get_done);
enable := F_TRIG.Q;
END_PROGRAM

PROGRAM INI_PARSER_BUF_DEMO
  VAR
    STATION_NAME : STRING;
    STATION_IP : STRING;
    SMTP_SERVER : STRING;
    SMTP_FROM : STRING;
    IPB : INI_PARSER_BUF;
    FS : FILE_SERVER;
    FSD : FILE_SERVER_DATA;
    PT : NETWORK_BUFFER;
    section : INT;
    key : STRING(OSCAT_BASIC.STRING_LENGTH);
    value : STRING(OSCAT_BASIC.STRING_LENGTH);
    str : STRING(OSCAT_BASIC.STRING_LENGTH);
    step : INT;
    result : BYTE;
    offset : UDINT;
    run : BYTE;
    done : BOOL;
  END_VAR

            (* Demo-Programm: INI-Datei mittels Enumeration auswerten *)

(* ----- den nachfolgenden Textblock als datei "config.ini" auf der sps ablegen ---
# Demo - Initialisierungsdatei

[Station]
NAME=Test_Station_1
IP=192.168.178.1

[SMTP]
SERVER=test.server.de
FROM=test1@gmx.net
---------------------------------------------------------------------------------*)

CASE step OF

00:	IF NOT done THEN
	 	(* File_Daten einrichten  *)
		FSD.FILENAME := 'config.ini'; (* Dateiname *)
		FSD.MODE := 1; (* vorhandene Datei zum lesen öffnen *)
		FSD.OFFSET := 0; (* Start bei Dateianfang *)
		PT.SIZE := 65535; (* maximale länge einlesen *)
		step := 10;
	END_IF;

10:	IF FSD.MODE = 0 THEN (* Datei geöffnet ? *)
		OFFSET := 0; (* Start Offset vorgeben *)
		str := '';
		run := 3; (* key suchen *)
		step := 20;
	END_IF;

20:	IF run = 0 THEN
		(* ---------------------- Debug-Message ----------------------------*)
		(*IF _debug_enable THEN
			LOG_CL.NEW_MSG := 'IPBD: /key >~1< /value >~2< /offset ~3 /Run ~4 /Result ~5';
			LOG_CL.PRINTF[1] := key;
			LOG_CL.PRINTF[2] := value;
			LOG_CL.PRINTF[3] := UDINT_TO_STRING(OFFSET);
			LOG_CL.PRINTF[4] := BYTE_TO_STRING(run);
			LOG_CL.PRINTF[5] := BYTE_TO_STRING(result);
			LOG_MSG();
		END_IF;*)
		(* -----------------------------------------------------------------*)

		run := 3; (* vorbelegung -> naechsten key suchen *)

		IF result = 1 THEN (* neue Sektion gefunden *)
			IF key = 'Station' THEN
				section := 1;
			ELSIF key = 'SMTP' THEN
				section := 2;

			(* hier können weitere Section hinzugefügt werden *)

			ELSE
				section := 0; (* unbekannte sektion gefunden -> ignorieren *)
			END_IF;

		ELSIF result = 2 AND section > 0 THEN (* Key in einer bekannten sektion gefunden *)

			CASE section OF

			1:  (* Section: Station *)
				IF key = 'NAME' THEN
					STATION_NAME := value; (* Name *)
				ELSIF key = 'IP' THEN
					STATION_IP := value; (* IP-Adresse *)
				END_IF;

				(* hier können weitere Schlüsselsauswertungen hinzugefügt werden *)

			2:  (* Section: SMTP *)
				IF key = 'SERVER' THEN
					SMTP_SERVER := value; (* SMTP Server *)
				ELSIF key = 'FROM' THEN
					SMTP_FROM := value; (* SMTP Absender *)
				END_IF;

				(* hier können weitere Schlüsselsauswertungen hinzugefügt werden *)

			END_CASE;

		ELSIF result = 10 THEN (* nichts mehr gefunden *)
			run := 0; (* keine weitere INI Auswertung erwünscht *)
			FSD.MODE := 5; (* Datei schliessen *)
			step := 30;
		END_IF;
	END_IF;

30:	IF FSD.MODE = 0 THEN (* Datei geschlossen ? *)
		step := 0;
		done := TRUE;
	END_IF;

END_CASE;

IPB(STR:=str,RUN:=run,OFFSET:=OFFSET,KEY:=key,VALUE:=value,PT:=PT); (* INI PARAMETER BUF *)
result:=IPB.RESULT;

FS(FSD:=FSD,PT:=PT); (* FILE_SERVER *)
          
END_PROGRAM

PROGRAM INI_PARSER_FILE_DEMO
  VAR
    STATION_NAME : STRING;
    STATION_IP : STRING;
    SMTP_SERVER : STRING;
    SMTP_FROM : STRING;
    IPF : INI_PARSER_FILE;
    FS : FILE_SERVER;
    FSD : FILE_SERVER_DATA;
    PT : NETWORK_BUFFER;
    section : INT;
    filename : STRING;
    key : STRING(OSCAT_BASIC.STRING_LENGTH);
    value : STRING(OSCAT_BASIC.STRING_LENGTH);
    str : STRING(OSCAT_BASIC.STRING_LENGTH);
    step : INT;
    result : BYTE;
    offset : UDINT;
    run : BYTE;
    done : BOOL;
  END_VAR

            (* Demo-Programm: INI-Datei mittels Enumeration auswerten *)

(* ----- den nachfolgenden Textblock als datei "config.ini" auf der sps ablegen ---
# Demo - Initialisierungsdatei

[Station]
NAME=Test_Station_1
IP=192.168.178.1

[SMTP]
SERVER=test.server.de
FROM=test1@gmx.net
---------------------------------------------------------------------------------*)

CASE step OF

00:	IF NOT done THEN
		filename := 'config.ini'; (* File_Daten einrichten *)
		OFFSET := 0; (* Start Offset vorgeben *)
		str := '';
		run := 3; (* key suchen *)
		step := 20;
	END_IF;

20:	IF run = 0 THEN (* kein Befehl mehr aktiv ? *)
		(* ---------------------- Debug-Message ----------------------------*)
		(*IF _debug_enable THEN
			LOG_CL.NEW_MSG := 'IPFD: /key >~1< /value >~2< /offset ~3 /Run ~4 /Result ~5';
			LOG_CL.PRINTF[1] := key;
			LOG_CL.PRINTF[2] := value;
			LOG_CL.PRINTF[3] := UDINT_TO_STRING(OFFSET);
			LOG_CL.PRINTF[4] := BYTE_TO_STRING(run);
			LOG_CL.PRINTF[5] := BYTE_TO_STRING(result);
			LOG_MSG();
		END_IF;*)
		(* -----------------------------------------------------------------*)

		run := 3; (* vorbelegung -> naechsten key suchen *)

		IF result = 1 THEN (* neue Sektion gefunden *)
			IF key = 'Station' THEN
				section := 1;
			ELSIF key = 'SMTP' THEN
				section := 2;

			(* hier können weitere Section hinzugefügt werden *)

			ELSE
				section := 0; (* unbekannte sektion gefunden -> ignorieren *)
			END_IF;

		ELSIF result = 2 AND section > 0 THEN (* Key in einer bekannten sektion gefunden *)

			CASE section OF

			1:  (* Section: Station *)
				IF key = 'NAME' THEN
					STATION_NAME := value; (* Name *)
				ELSIF key = 'IP' THEN
					STATION_IP := value; (* IP-Adresse *)
				END_IF;

				(* hier können weitere Schlüsselsauswertungen hinzugefügt werden *)

			2:  (* Section: SMTP *)
				IF key = 'SERVER' THEN
					SMTP_SERVER := value; (* SMTP Server *)
				ELSIF key = 'FROM' THEN
					SMTP_FROM := value; (* SMTP Absender *)
				END_IF;

				(* hier können weitere Schlüsselsauswertungen hinzugefügt werden *)

			END_CASE;

		ELSIF result = 10 THEN (* nichts mehr gefunden *)
			run := 0; (* keine weitere INI Auswertung erwünscht *)
			FSD.MODE := 5; (* Datei schliessen *)
			step := 30;
		END_IF;
	END_IF;

30:	IF FSD.MODE = 0 THEN (* Befehl Datei schliessen beendet *)
		step := 0;
		done := TRUE;
	END_IF;

END_CASE;

IPF(FILENAME:=FILENAME,FSD:=FSD,STR:=str,RUN:=run,OFFSET:=OFFSET,KEY:=key,VALUE:=value,PT:=PT); (* INI PARAMETER FILE *)
result:=IPF.RESULT;

FS(FSD:=FSD,PT:=PT); (* FILE_SERVER *)
          
END_PROGRAM

PROGRAM IP2GEO_DEMO
  VAR
    IP_C : IP_C;
    S_BUF : NETWORK_BUFFER;
    R_BUF : NETWORK_BUFFER;
    IP_CONTROL_1 : IP_CONTROL;
    CLK_PRG : oscat_basic.CLK_PRG;
    IP2GEO_1 : IP2GEO;
    GEO : IP2GEO_DATA;
    activate : BOOL := TRUE;
    done : BOOL;
    busy : BOOL;
    error_c : DWORD;
    error_t : BYTE;
  END_VAR

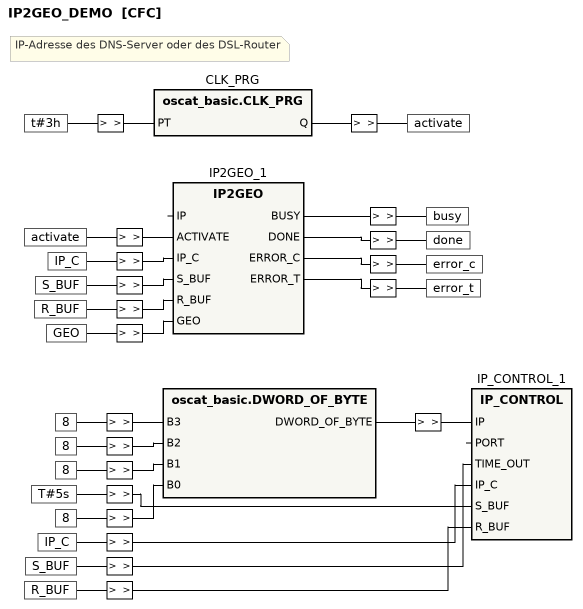
(* CFC diagram, written out as Structured Text *)
CLK_PRG(PT := t#3h);
activate := CLK_PRG.Q;
IP2GEO_1(ACTIVATE := activate, IP_C := IP_C, S_BUF := S_BUF, R_BUF := R_BUF, GEO := GEO);
busy := IP2GEO_1.BUSY;
done := IP2GEO_1.DONE;
error_c := IP2GEO_1.ERROR_C;
error_t := IP2GEO_1.ERROR_T;
(* IP-Adresse des DNS-Server oder des DSL-Router *)
IP_CONTROL_1(IP := oscat_basic.DWORD_OF_BYTE(8, 8, 8, 8), TIME_OUT := T#5s, IP_C := IP_C, S_BUF := S_BUF, R_BUF := R_BUF);
END_PROGRAM

PROGRAM IRTRANS_DEMO
  VAR
    IP_C : IP_C;
    S_BUF : NETWORK_BUFFER_SHORT;
    R_BUF : NETWORK_BUFFER_SHORT;
    IP_CONTROL2 : IP_CONTROL2;
    IRTRANS_DECODE : IRTRANS_DECODE;
    IRTRANS_RCV_4 : IRTRANS_RCV_4;
    DRIVER_4 : oscat_basic.DRIVER_4;
    IRTRANS_SERVER : IRTRANS_SERVER;
    IRTRANS_SND_8_1 : IRTRANS_SND_8;
    IRTRANS_SND_8_2 : IRTRANS_SND_8;
    Q0 : BOOL;
    Q1 : BOOL;
    Q2 : BOOL;
    Q3 : BOOL;
    error : BOOL;
    error_server : DWORD;
    Send_1_0 : BOOL := TRUE;
    Send_1_1 : BOOL;
    Send_1_2 : BOOL;
    Send_1_3 : BOOL;
    Send_1_4 : BOOL;
    Send_1_5 : BOOL;
    Send_1_6 : BOOL;
    Send_1_7 : BOOL;
    Send_2_0 : BOOL := TRUE;
    Send_2_1 : BOOL;
    Send_2_2 : BOOL;
    Send_2_3 : BOOL;
    Send_2_4 : BOOL;
    Send_2_5 : BOOL;
    Send_2_6 : BOOL;
    Send_2_7 : BOOL;
    R_ENABLE : BOOL;
    S_ENABLE : BOOL;
    MODE : BOOL := FALSE;
    KEY_1 : BYTE;
    KEY_2 : BYTE;
  END_VAR

(* CFC diagram, written out as Structured Text *)
(* IRTRANS Empfang *)
IRTRANS_DECODE(IP_C := IP_C, R_BUF := R_BUF);
(* IRTRANS Senden (beliebig viele Instanzen zulässig !) *)
error := IRTRANS_DECODE.ERROR;
IRTRANS_RCV_4(CMD := IRTRANS_DECODE.CMD, DEV := IRTRANS_DECODE.DEV, KEY := IRTRANS_DECODE.KEY);
DRIVER_4(IN0 := IRTRANS_RCV_4.Q0, IN1 := IRTRANS_RCV_4.Q1, IN2 := IRTRANS_RCV_4.Q2, IN3 := IRTRANS_RCV_4.Q3);
Q0 := DRIVER_4.Q0;
Q1 := DRIVER_4.Q1;
Q2 := DRIVER_4.Q2;
Q3 := DRIVER_4.Q3;
KEY_1 := IRTRANS_SND_8_1.KEY;
KEY_2 := IRTRANS_SND_8_2.KEY;
(* Hardwareneutraler Ethernet IP *)
(* IRTRANS Kommunikation *)
IRTRANS_SERVER(UDP_TCP := MODE, IP_C := IP_C, S_BUF := S_BUF, R_BUF := R_BUF);
S_ENABLE := IRTRANS_SERVER.S_ENABLE;
R_ENABLE := IRTRANS_SERVER.R_ENABLE;
error_server := IRTRANS_SERVER.ERROR;
IP_CONTROL2(PORT := 21000, TIME_OUT := T#2s, IP_C := IP_C, S_BUF := S_BUF, R_BUF := R_BUF);
IRTRANS_SND_8_2(IN_0 := Send_2_0, IN_1 := Send_2_1, IN_2 := Send_2_2, IN_3 := Send_2_3, IN_4 := Send_2_4, IN_5 := Send_2_5, IN_6 := Send_2_6, IN_7 := Send_2_7, T_REPEAT := T#500ms, IP_C := IP_C, S_BUF := S_BUF);
IRTRANS_SND_8_1(IN_0 := Send_1_0, IN_1 := Send_1_1, IN_2 := Send_1_2, IN_3 := Send_1_3, IN_4 := Send_1_4, IN_5 := Send_1_5, IN_6 := Send_1_6, IN_7 := Send_1_7, T_REPEAT := T#500ms, IP_C := IP_C, S_BUF := S_BUF);
END_PROGRAM

PROGRAM MB_CLIENT_DEMO
  VAR
    IP_CONTROL2_1 : IP_CONTROL2;
    MB_CLIENT_1 : MB_CLIENT;
    IP_C : IP_C;
    S_BUF : NETWORK_BUFFER_SHORT;
    R_BUF : NETWORK_BUFFER_SHORT;
    DATA : ARRAY[0..255] OF WORD;
    W_DATA_BITPOS : INT;
    W_DATA_ADR : INT;
    W_POINTS : INT;
    W_ADDR : INT;
    R_DATA_BITPOS : INT;
    R_DATA_ADR : INT;
    R_POINTS : INT;
    R_ADDR : INT;
    FC : INT;
    ENABLE : BOOL;
  END_VAR

(* CFC diagram, written out as Structured Text *)
MB_CLIENT_1(DATA_SIZE := 256, ENABLE := ENABLE, UDP := FALSE, FC := FC, UNIT_ID := 3, R_ADDR := R_ADDR, R_POINTS := R_POINTS, R_DATA_ADR := R_DATA_ADR, R_DATA_BITPOS := R_DATA_BITPOS, W_ADDR := W_ADDR, W_POINTS := W_POINTS, W_DATA_ADR := W_DATA_ADR, W_DATA_BITPOS := W_DATA_BITPOS, DELAY := T#1s, IP_C := IP_C, S_BUF := S_BUF, R_BUF := R_BUF, DATA := DATA);
(* IP-Adresse des MODBUS-TCP-Server *)
IP_CONTROL2_1(IP := oscat_basic.DWORD_OF_BYTE(192, 168, 178, 001), PORT := 502, TIME_OUT := T#5s, IP_C := IP_C, S_BUF := S_BUF, R_BUF := R_BUF);
END_PROGRAM

PROGRAM MB_SERVER_DEMO
  VAR
    IP_CONTROL2_1 : IP_CONTROL2;
    MB_SERVER_1 : MB_SERVER;
    IP_C : IP_C;
    S_BUF : NETWORK_BUFFER_SHORT;
    R_BUF : NETWORK_BUFFER_SHORT;
    DATA : ARRAY[0..255] OF WORD;
    VMAP : ARRAY[1..10] OF VMAP_DATA;
    error : DWORD;
  END_VAR

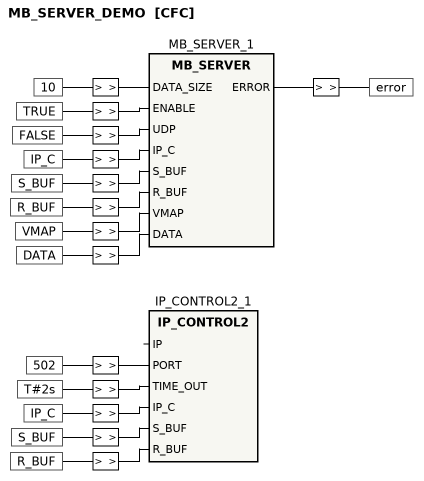
(* CFC diagram, written out as Structured Text *)
MB_SERVER_1(DATA_SIZE := 10, ENABLE := TRUE, UDP := FALSE, IP_C := IP_C, S_BUF := S_BUF, R_BUF := R_BUF, VMAP := VMAP, DATA := DATA);
IP_CONTROL2_1(PORT := 502, TIME_OUT := T#2s, IP_C := IP_C, S_BUF := S_BUF, R_BUF := R_BUF);
error := MB_SERVER_1.ERROR;
END_PROGRAM

PROGRAM MD5_CRAM_AUTH_DEMO
  VAR
    run : BOOL := TRUE;
    timestamp : STRING(64) := 'PDQwMzYuMTA3NjMyNDM4MUBndWlsZGVuc3Rlcm4uemVpdGZvcm0uZGU+';
    password : STRING := 'geheimes_passwort';
    username : STRING := 'benutzer@zeitform.de';
    auth_key : STRING(OSCAT_BASIC.STRING_LENGTH);
    MD5_CRAM_AUTH : MD5_CRAM_AUTH;
  END_VAR

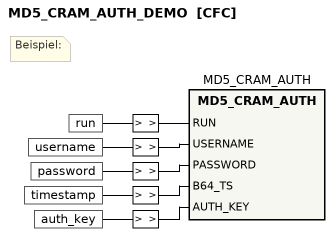
(* CFC diagram, written out as Structured Text *)
(* Beispiel: *)
MD5_CRAM_AUTH(RUN := run, USERNAME := username, PASSWORD := password, B64_TS := timestamp, AUTH_KEY := auth_key);
END_PROGRAM

PROGRAM NET_VAR_MASTER_DEMO
  VAR
    NET_VAR_CONTROL_1 : NET_VAR_CONTROL;
    activate : BOOL := TRUE;
    run : BOOL;
    udp : BOOL := TRUE;
    master : BOOL := TRUE;
    remote_port : WORD := 10000;
    scan_time : TIME := TIME#1s0ms;
    watchdog : TIME := TIME#2s0ms;
    error : DWORD;
    x : NET_VAR_DATA;
    NET_VAR_BOOL8_1 : NET_VAR_BOOL8;
    id_b8 : BYTE;
    in_b1 : BOOL;
    in_b2 : BOOL;
    in_b3 : BOOL;
    in_b4 : BOOL;
    in_b5 : BOOL;
    in_b6 : BOOL;
    in_b7 : BOOL;
    in_b8 : BOOL;
    out_b1 : BOOL;
    out_b2 : BOOL;
    out_b3 : BOOL;
    out_b4 : BOOL;
    out_b5 : BOOL;
    out_b6 : BOOL;
    out_b7 : BOOL;
    out_b8 : BOOL;
    NET_VAR_STRING_1 : NET_VAR_STRING;
    in_s1 : STRING(OSCAT_BASIC.STRING_LENGTH);
    out_s1 : STRING(OSCAT_BASIC.STRING_LENGTH);
    id_s : BYTE;
    NET_VAR_BUFFER_1 : NET_VAR_BUFFER;
    id_bu : BYTE;
    BUF_IN : ARRAY[1..64] OF BYTE;
    BUF_OUT : ARRAY[1..64] OF BYTE;
    id_dw : BYTE;
    NET_VAR_DWORD8_1 : NET_VAR_DWORD8;
    in_dw1 : DWORD;
    in_dw2 : DWORD;
    in_dw3 : DWORD;
    in_dw4 : DWORD;
    in_dw5 : DWORD;
    in_dw6 : DWORD;
    in_dw7 : DWORD;
    in_dw8 : DWORD;
    out_dw1 : DWORD;
    out_dw2 : DWORD;
    out_dw3 : DWORD;
    out_dw4 : DWORD;
    out_dw5 : DWORD;
    out_dw6 : DWORD;
    out_dw7 : DWORD;
    out_dw8 : DWORD;
    NET_VAR_REAL8_1 : NET_VAR_REAL8;
    in_r1 : REAL;
    in_r2 : REAL;
    in_r3 : REAL;
    in_r4 : REAL;
    in_r5 : REAL;
    in_r6 : REAL;
    in_r7 : REAL;
    in_r8 : REAL;
    out_r1 : REAL;
    out_r2 : REAL;
    out_r3 : REAL;
    out_r4 : REAL;
    out_r5 : REAL;
    out_r6 : REAL;
    out_r7 : REAL;
    out_r8 : REAL;
    id_r : BYTE;
    NET_VAR_X8_1 : NET_VAR_X8;
    in_x_re1 : REAL;
    in_x_re2 : REAL;
    in_x_di1 : DINT;
    in_x_di2 : DINT;
    in_x_ud1 : UDINT;
    in_x_ud2 : UDINT;
    in_x_dw1 : DWORD;
    in_x_dw2 : DWORD;
    out_x_re1 : REAL;
    out_x_re2 : REAL;
    out_x_di1 : DINT;
    out_x_di2 : DINT;
    out_x_ud1 : UDINT;
    out_x_ud2 : UDINT;
    out_x_dw1 : DWORD;
    out_x_dw2 : DWORD;
    id_x8 : BYTE;
  END_VAR

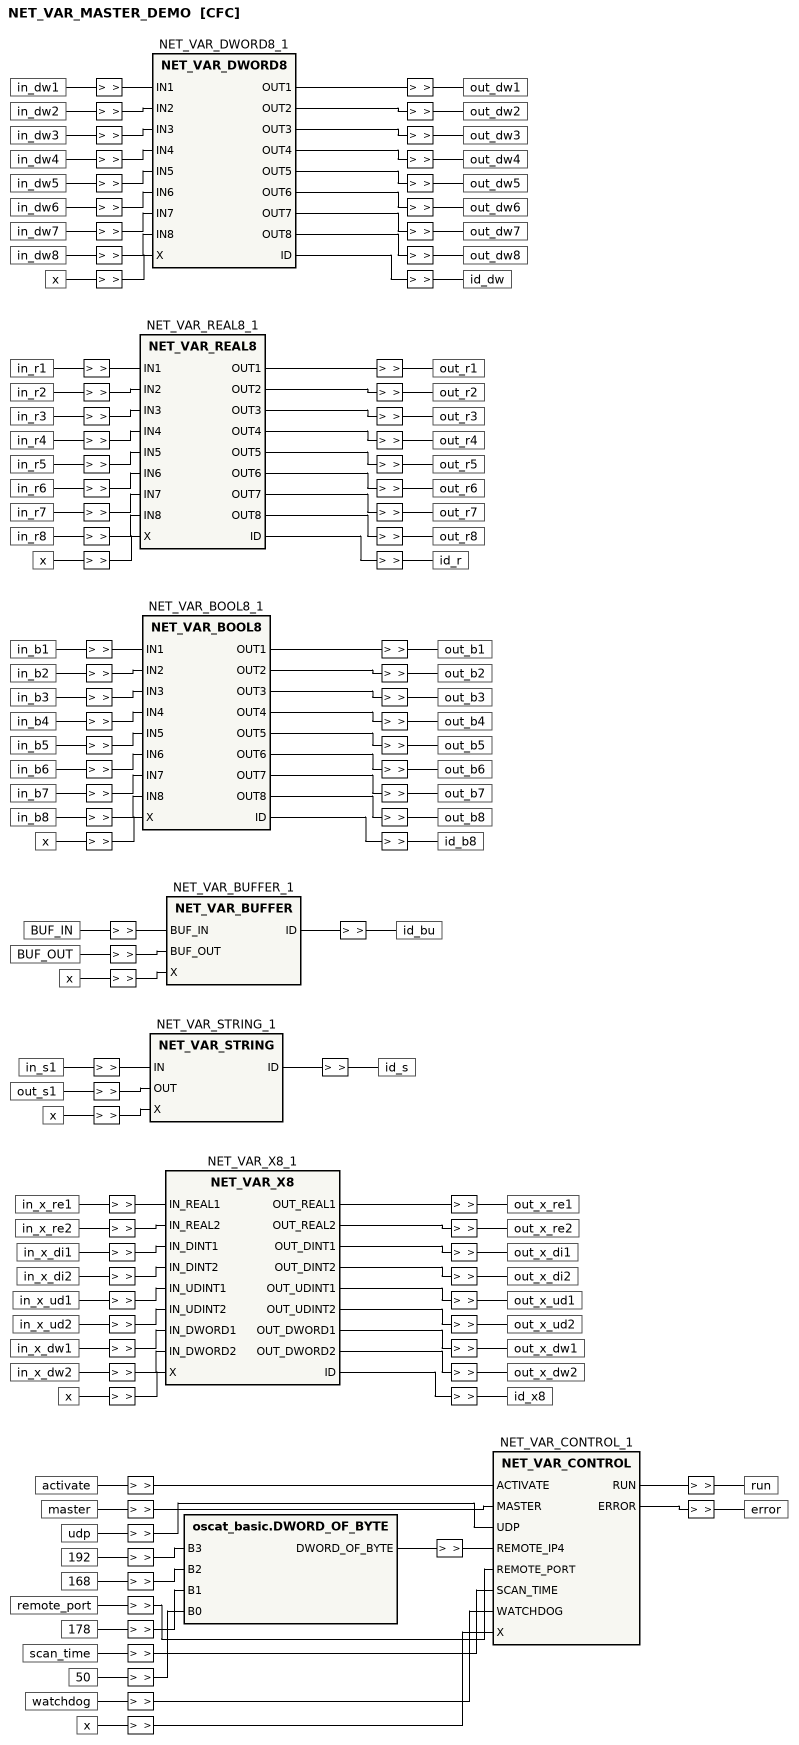
(* CFC diagram, written out as Structured Text *)
NET_VAR_DWORD8_1(IN1 := in_dw1, IN2 := in_dw2, IN3 := in_dw3, IN4 := in_dw4, IN5 := in_dw5, IN6 := in_dw6, IN7 := in_dw7, IN8 := in_dw8, X := x);
out_dw1 := NET_VAR_DWORD8_1.OUT1;
out_dw2 := NET_VAR_DWORD8_1.OUT2;
out_dw3 := NET_VAR_DWORD8_1.OUT3;
out_dw4 := NET_VAR_DWORD8_1.OUT4;
out_dw5 := NET_VAR_DWORD8_1.OUT5;
out_dw6 := NET_VAR_DWORD8_1.OUT6;
out_dw7 := NET_VAR_DWORD8_1.OUT7;
out_dw8 := NET_VAR_DWORD8_1.OUT8;
id_dw := NET_VAR_DWORD8_1.ID;
NET_VAR_REAL8_1(IN1 := in_r1, IN2 := in_r2, IN3 := in_r3, IN4 := in_r4, IN5 := in_r5, IN6 := in_r6, IN7 := in_r7, IN8 := in_r8, X := x);
out_r1 := NET_VAR_REAL8_1.OUT1;
out_r2 := NET_VAR_REAL8_1.OUT2;
out_r3 := NET_VAR_REAL8_1.OUT3;
out_r4 := NET_VAR_REAL8_1.OUT4;
out_r5 := NET_VAR_REAL8_1.OUT5;
out_r6 := NET_VAR_REAL8_1.OUT6;
out_r7 := NET_VAR_REAL8_1.OUT7;
out_r8 := NET_VAR_REAL8_1.OUT8;
id_r := NET_VAR_REAL8_1.ID;
NET_VAR_BOOL8_1(IN1 := in_b1, IN2 := in_b2, IN3 := in_b3, IN4 := in_b4, IN5 := in_b5, IN6 := in_b6, IN7 := in_b7, IN8 := in_b8, X := x);
out_b1 := NET_VAR_BOOL8_1.OUT1;
out_b2 := NET_VAR_BOOL8_1.OUT2;
out_b3 := NET_VAR_BOOL8_1.OUT3;
out_b4 := NET_VAR_BOOL8_1.OUT4;
out_b5 := NET_VAR_BOOL8_1.OUT5;
out_b6 := NET_VAR_BOOL8_1.OUT6;
out_b7 := NET_VAR_BOOL8_1.OUT7;
out_b8 := NET_VAR_BOOL8_1.OUT8;
id_b8 := NET_VAR_BOOL8_1.ID;
NET_VAR_BUFFER_1(BUF_IN := BUF_IN, BUF_OUT := BUF_OUT, X := x);
id_bu := NET_VAR_BUFFER_1.ID;
NET_VAR_STRING_1(IN := in_s1, OUT := out_s1, X := x);
id_s := NET_VAR_STRING_1.ID;
NET_VAR_X8_1(IN_REAL1 := in_x_re1, IN_REAL2 := in_x_re2, IN_DINT1 := in_x_di1, IN_DINT2 := in_x_di2, IN_UDINT1 := in_x_ud1, IN_UDINT2 := in_x_ud2, IN_DWORD1 := in_x_dw1, IN_DWORD2 := in_x_dw2, X := x);
out_x_re1 := NET_VAR_X8_1.OUT_REAL1;
out_x_re2 := NET_VAR_X8_1.OUT_REAL2;
out_x_di1 := NET_VAR_X8_1.OUT_DINT1;
out_x_di2 := NET_VAR_X8_1.OUT_DINT2;
out_x_ud1 := NET_VAR_X8_1.OUT_UDINT1;
out_x_ud2 := NET_VAR_X8_1.OUT_UDINT2;
out_x_dw1 := NET_VAR_X8_1.OUT_DWORD1;
out_x_dw2 := NET_VAR_X8_1.OUT_DWORD2;
id_x8 := NET_VAR_X8_1.ID;
NET_VAR_CONTROL_1(ACTIVATE := activate, MASTER := master, UDP := udp, REMOTE_IP4 := oscat_basic.DWORD_OF_BYTE(192, 168, 178, 50), REMOTE_PORT := remote_port, SCAN_TIME := scan_time, WATCHDOG := watchdog, X := x);
run := NET_VAR_CONTROL_1.RUN;
error := NET_VAR_CONTROL_1.ERROR;
END_PROGRAM

PROGRAM NET_VAR_SLAVE_DEMO
  VAR
    NET_VAR_CONTROL_1 : NET_VAR_CONTROL;
    activate : BOOL := TRUE;
    run : BOOL;
    udp : BOOL := TRUE;
    master : BOOL := FALSE;
    remote_port : WORD := 10000;
    scan_time : TIME := TIME#1s0ms;
    watchdog : TIME := TIME#2s0ms;
    error : DWORD;
    x : NET_VAR_DATA;
    NET_VAR_BOOL8_1 : NET_VAR_BOOL8;
    id_b8 : BYTE;
    in_b1 : BOOL;
    in_b2 : BOOL;
    in_b3 : BOOL;
    in_b4 : BOOL;
    in_b5 : BOOL;
    in_b6 : BOOL;
    in_b7 : BOOL;
    in_b8 : BOOL;
    out_b1 : BOOL;
    out_b2 : BOOL;
    out_b3 : BOOL;
    out_b4 : BOOL;
    out_b5 : BOOL;
    out_b6 : BOOL;
    out_b7 : BOOL;
    out_b8 : BOOL;
    NET_VAR_STRING_1 : NET_VAR_STRING;
    in_s1 : STRING(OSCAT_BASIC.STRING_LENGTH);
    out_s1 : STRING(OSCAT_BASIC.STRING_LENGTH);
    id_s : BYTE;
    NET_VAR_BUFFER_1 : NET_VAR_BUFFER;
    id_bu : BYTE;
    BUF_IN : ARRAY[1..64] OF BYTE;
    BUF_OUT : ARRAY[1..64] OF BYTE;
    id_dw : BYTE;
    NET_VAR_DWORD8_1 : NET_VAR_DWORD8;
    in_dw1 : DWORD;
    in_dw2 : DWORD;
    in_dw3 : DWORD;
    in_dw4 : DWORD;
    in_dw5 : DWORD;
    in_dw6 : DWORD;
    in_dw7 : DWORD;
    in_dw8 : DWORD;
    out_dw1 : DWORD;
    out_dw2 : DWORD;
    out_dw3 : DWORD;
    out_dw4 : DWORD;
    out_dw5 : DWORD;
    out_dw6 : DWORD;
    out_dw7 : DWORD;
    out_dw8 : DWORD;
    NET_VAR_REAL8_1 : NET_VAR_REAL8;
    in_r1 : REAL;
    in_r2 : REAL;
    in_r3 : REAL;
    in_r4 : REAL;
    in_r5 : REAL;
    in_r6 : REAL;
    in_r7 : REAL;
    in_r8 : REAL;
    out_r1 : REAL;
    out_r2 : REAL;
    out_r3 : REAL;
    out_r4 : REAL;
    out_r5 : REAL;
    out_r6 : REAL;
    out_r7 : REAL;
    out_r8 : REAL;
    id_r : BYTE;
    NET_VAR_X8_1 : NET_VAR_X8;
    in_x_re1 : REAL;
    in_x_re2 : REAL;
    in_x_di1 : DINT;
    in_x_di2 : DINT;
    in_x_ud1 : UDINT;
    in_x_ud2 : UDINT;
    in_x_dw1 : DWORD;
    in_x_dw2 : DWORD;
    out_x_re1 : REAL;
    out_x_re2 : REAL;
    out_x_di1 : DINT;
    out_x_di2 : DINT;
    out_x_ud1 : UDINT;
    out_x_ud2 : UDINT;
    out_x_dw1 : DWORD;
    out_x_dw2 : DWORD;
    id_x8 : BYTE;
  END_VAR

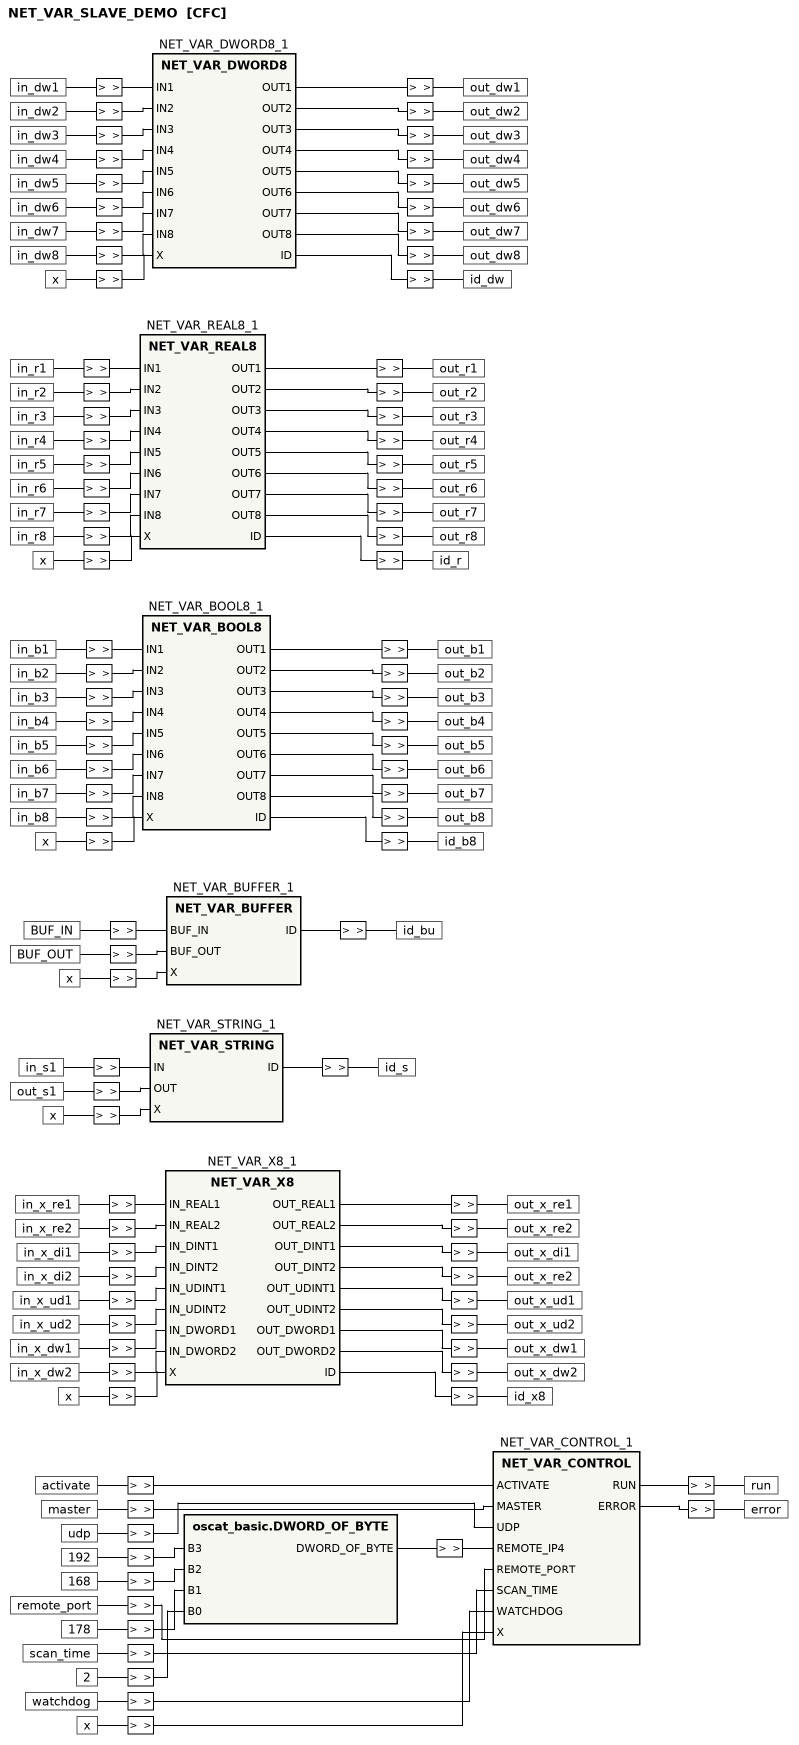
(* CFC diagram, written out as Structured Text *)
NET_VAR_DWORD8_1(IN1 := in_dw1, IN2 := in_dw2, IN3 := in_dw3, IN4 := in_dw4, IN5 := in_dw5, IN6 := in_dw6, IN7 := in_dw7, IN8 := in_dw8, X := x);
out_dw1 := NET_VAR_DWORD8_1.OUT1;
out_dw2 := NET_VAR_DWORD8_1.OUT2;
out_dw3 := NET_VAR_DWORD8_1.OUT3;
out_dw4 := NET_VAR_DWORD8_1.OUT4;
out_dw5 := NET_VAR_DWORD8_1.OUT5;
out_dw6 := NET_VAR_DWORD8_1.OUT6;
out_dw7 := NET_VAR_DWORD8_1.OUT7;
out_dw8 := NET_VAR_DWORD8_1.OUT8;
id_dw := NET_VAR_DWORD8_1.ID;
NET_VAR_REAL8_1(IN1 := in_r1, IN2 := in_r2, IN3 := in_r3, IN4 := in_r4, IN5 := in_r5, IN6 := in_r6, IN7 := in_r7, IN8 := in_r8, X := x);
out_r1 := NET_VAR_REAL8_1.OUT1;
out_r2 := NET_VAR_REAL8_1.OUT2;
out_r3 := NET_VAR_REAL8_1.OUT3;
out_r4 := NET_VAR_REAL8_1.OUT4;
out_r5 := NET_VAR_REAL8_1.OUT5;
out_r6 := NET_VAR_REAL8_1.OUT6;
out_r7 := NET_VAR_REAL8_1.OUT7;
out_r8 := NET_VAR_REAL8_1.OUT8;
id_r := NET_VAR_REAL8_1.ID;
NET_VAR_BOOL8_1(IN1 := in_b1, IN2 := in_b2, IN3 := in_b3, IN4 := in_b4, IN5 := in_b5, IN6 := in_b6, IN7 := in_b7, IN8 := in_b8, X := x);
out_b1 := NET_VAR_BOOL8_1.OUT1;
out_b2 := NET_VAR_BOOL8_1.OUT2;
out_b3 := NET_VAR_BOOL8_1.OUT3;
out_b4 := NET_VAR_BOOL8_1.OUT4;
out_b5 := NET_VAR_BOOL8_1.OUT5;
out_b6 := NET_VAR_BOOL8_1.OUT6;
out_b7 := NET_VAR_BOOL8_1.OUT7;
out_b8 := NET_VAR_BOOL8_1.OUT8;
id_b8 := NET_VAR_BOOL8_1.ID;
NET_VAR_BUFFER_1(BUF_IN := BUF_IN, BUF_OUT := BUF_OUT, X := x);
id_bu := NET_VAR_BUFFER_1.ID;
NET_VAR_STRING_1(IN := in_s1, OUT := out_s1, X := x);
id_s := NET_VAR_STRING_1.ID;
NET_VAR_X8_1(IN_REAL1 := in_x_re1, IN_REAL2 := in_x_re2, IN_DINT1 := in_x_di1, IN_DINT2 := in_x_di2, IN_UDINT1 := in_x_ud1, IN_UDINT2 := in_x_ud2, IN_DWORD1 := in_x_dw1, IN_DWORD2 := in_x_dw2, X := x);
out_x_re1 := NET_VAR_X8_1.OUT_REAL1;
out_x_re2 := NET_VAR_X8_1.OUT_REAL2;
out_x_di1 := NET_VAR_X8_1.OUT_DINT1;
out_x_re2 := NET_VAR_X8_1.OUT_DINT2;
out_x_ud1 := NET_VAR_X8_1.OUT_UDINT1;
out_x_ud2 := NET_VAR_X8_1.OUT_UDINT2;
out_x_dw1 := NET_VAR_X8_1.OUT_DWORD1;
out_x_dw2 := NET_VAR_X8_1.OUT_DWORD2;
id_x8 := NET_VAR_X8_1.ID;
NET_VAR_CONTROL_1(ACTIVATE := activate, MASTER := master, UDP := udp, REMOTE_IP4 := oscat_basic.DWORD_OF_BYTE(192, 168, 178, 2), REMOTE_PORT := remote_port, SCAN_TIME := scan_time, WATCHDOG := watchdog, X := x);
run := NET_VAR_CONTROL_1.RUN;
error := NET_VAR_CONTROL_1.ERROR;
END_PROGRAM

PROGRAM RC4_CRYPT_DEMO
  VAR
    RC4_CRYPT_STREAM : RC4_CRYPT_STREAM;
    buf : ARRAY[0..63] OF BYTE := [110, 60, 3, 219];  (* crypt *)
    mode : INT;
    key : STRING := '1234';
    size : UDINT := 4;
    pos : UDINT;
  END_VAR

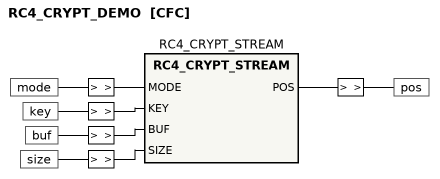
(* CFC diagram, written out as Structured Text *)
RC4_CRYPT_STREAM(MODE := mode, KEY := key, BUF := buf, SIZE := size);
pos := RC4_CRYPT_STREAM.POS;
END_PROGRAM

PROGRAM SHA1_MD5_DEMO
  VAR
    text : STRING(OSCAT_BASIC.STRING_LENGTH) := '<4036.1076324381@guildenstern.zeitform.de>';
    MD5_STR : MD5_STR;
    SHA1_STR : SHA1_STR;
    md5_hash : ARRAY[0..15] OF BYTE;
    sha1_hash : ARRAY[0..19] OF BYTE;
    start1 : BOOL := TRUE;
    start2 : BOOL := TRUE;
    done1 : BOOL;
    done2 : BOOL;
    md5_strh : STRING(32);
    sha1_strh : STRING(40);
  END_VAR

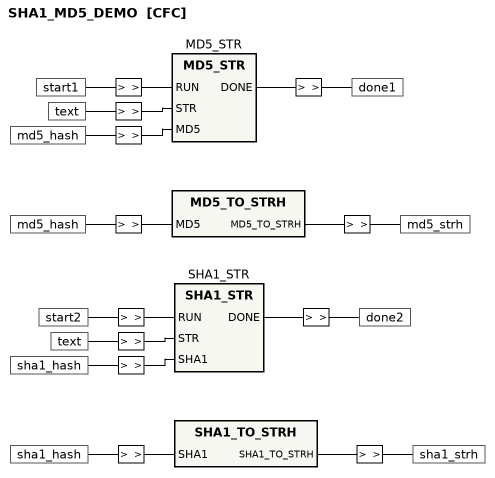
(* CFC diagram, written out as Structured Text *)
MD5_STR(RUN := start1, STR := text, MD5 := md5_hash);
done1 := MD5_STR.DONE;
md5_strh := MD5_TO_STRH(md5_hash);
SHA1_STR(RUN := start2, STR := text, SHA1 := sha1_hash);
done2 := SHA1_STR.DONE;
sha1_strh := SHA1_TO_STRH(sha1_hash);
END_PROGRAM

PROGRAM SMTP_CLIENT_DEMO
  VAR
    SMTP_CLIENT : SMTP_CLIENT;  (* smtp_server: STRING := 'oscat_test%freenet.de:oscat123456@mx.freenet.de'; smtp_mailfrom: STRING := 'oscat_test@freenet.de'; *)
    smtp_activate : BOOL;
    smtp_timeout : TIME := TIME#30s0ms;
    smtp_error_t : BYTE;
    smtp_error_c : DWORD;
    smtp_busy : BOOL;
    smtp_done : BOOL;
    smtp_dti : DT;
    smtp_dti_offset : INT := 60;
    smtp_files : STRING(OSCAT_BASIC.STRING_LENGTH) := '';
    smtp_server : STRING := '110876022:oscat123456@mail.gmx.net';
    smtp_mailfrom : STRING := 'oscat@gmx.net;Station_01';
    smtp_mailto : STRING(OSCAT_BASIC.STRING_LENGTH) := 'oscat@gmx.net';
    smtp_subject : STRING := 'Das ist der Betreff';
    smtp_body : STRING(OSCAT_BASIC.STRING_LENGTH) := 'Das ist der Email-Text';
  END_VAR

